KUKA KRL program: EPS_2_251806_MH02A_A_20260212042229.src

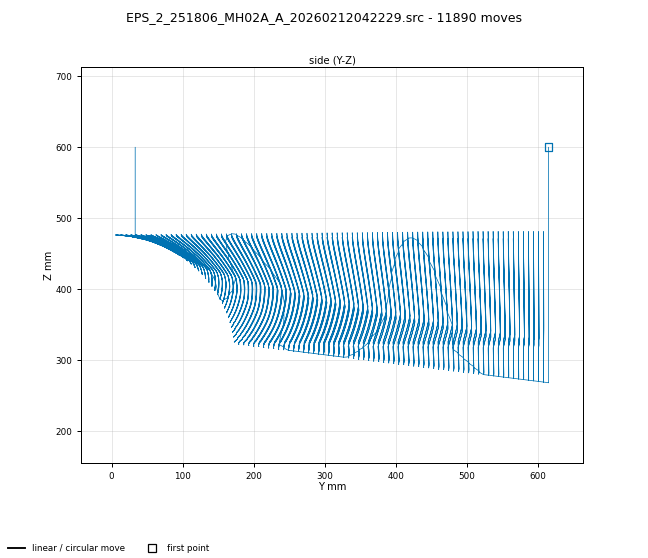
[picture p0: tool path of EPS_2_251806_MH02A_A_20260212042229.src, 11890 of 11892 moves have a stored position in this frame; points joined in program order, loops and branches not executed]
&ACCESS RVP
&REL 4
&COMMENT QRS 19112012
&PARAM EDITMASK = *
DEF PART()
EXT BAS (BAS_COMMAND :IN,REAL :IN )
INT I
BAS (#INITMOV,0 )

;KUKA QRS Post kuka4.cps  Date:22-06-2017 !

File_ID=3010

QRS_PRE_INIT()

;Init var - Until changes are made in qrs_pre_init
Outlet_Square_prg=0
Inlet_1_Square_prg=0
Inlet_2_Square_prg=0
Inlet_3_Square_prg=0
Inlet_4_Square_prg=0
Inlet_5_Square_prg=0

Outlet_1={X 0.000, Y 513.880, Z 332.000, B 0.000, E1 0.000 }
Inlet_1={X 0.000, Y 514.620, Z 322.000, B 0.000, E1 180.000 }
Outlet_1_type=299
Inlet_1_type=299
;QRS#1=Sidecore dimensions
;QRS#2=300-12" PVC SDR 35
;QRS#3=300-12" PVC SDR 35
;QRS#4=
;QRS#5=
;QRS#6=
;QRS#7=
;QRS#8=
;QRS#9=16M PSX
;QRS#10=16M PSX
;QRS#11=
;QRS#12=
;QRS#13=
;QRS#14=
;QRS#15=
;QRS#16=1220x127x762 2,5'
;QRS#17=EPS Height
;QRS#18=481,5
;QRS#19=*
;QRS#20= UPDATED VERSION 22-06-2017
;QRS#21=*
Outlet_Square=0150
Inlet_1_Square=0150
Inlet_2_Square=0
Inlet_3_Square=0
Inlet_4_Square=0
Inlet_5_Square=0
Mill_Square=1
Outlet_Square_Prg=206
Inlet_1_Square_prg=206

QRS_INIT()

$ADVANCE=5

; T1
PTP {E1 173.624,E2 173.624}
PTP {X 0,Y 615.47,A -85,B 0,C 180,E1 173.624,E2 173.624,E3 0,E4 0,E5 0,E6 0}
QRS_SPEED_INIT()
LIN {X 0,Y 615.47,Z 600,A -85,B 0,C 180,E1 173.624,E2 173.624,E3 0,E4 0,E5 0,E6 0} C_VEL
LIN {X 0,Y 615.47,Z 278.503,A -85,B 0,C 180,E1 173.624,E2 173.624} C_VEL
LIN {X 0,Y 615.47,Z 270.325,A -85,B 0,C 180,E1 173.624,E2 173.624} C_VEL
LIN {X 0,Y 615.455,Z 268.325,A -85,B 0,C 180,E1 173.438,E2 173.438} C_VEL
LIN {X 0,Y 615.494,Z 268.326,A -85,B 0,C 180,E1 170.801,E2 170.801} C_VEL
LIN {X 0,Y 615.492,Z 268.318,A -85,B 0,C 180,E1 168.139,E2 168.139} C_VEL
LIN {X 0,Y 615.446,Z 268.325,A -85,B 0,C 180,E1 165.45,E2 165.45} C_VEL
LIN {X 0,Y 615.486,Z 268.318,A -85,B 0,C 180,E1 162.729,E2 162.729} C_VEL
LIN {X 0,Y 615.479,Z 268.326,A -85,B 0,C 180,E1 159.967,E2 159.967} C_VEL
LIN {X 0,Y 615.454,Z 268.324,A -85,B 0,C 180,E1 157.659,E2 157.659} C_VEL
LIN {X 0,Y 615.479,Z 268.319,A -85,B 0,C 180,E1 155.008,E2 155.008} C_VEL
LIN {X 0,Y 615.46,Z 268.325,A -85,B 0,C 180,E1 152.083,E2 152.083} C_VEL
LIN {X 0,Y 615.467,Z 268.322,A -85,B 0,C 180,E1 149.839,E2 149.839} C_VEL
LIN {X 0,Y 615.476,Z 268.322,A -85,B 0,C 180,E1 147.542,E2 147.542} C_VEL
LIN {X 0,Y 615.46,Z 268.325,A -85,B 0,C 180,E1 145.183,E2 145.183} C_VEL
LIN {X 0,Y 615.492,Z 268.316,A -85,B 0,C 180,E1 142.758,E2 142.758} C_VEL
LIN {X 0,Y 615.472,Z 268.324,A -85,B 0,C 180,E1 139.911,E2 139.911} C_VEL
LIN {X 0,Y 615.453,Z 268.325,A -85,B 0,C 180,E1 137.644,E2 137.644} C_VEL
LIN {X 0,Y 615.491,Z 268.315,A -85,B 0,C 180,E1 134.932,E2 134.932} C_VEL
LIN {X 0,Y 615.455,Z 268.324,A -85,B 0,C 180,E1 132.077,E2 132.077} C_VEL
LIN {X 0,Y 615.486,Z 268.547,A -85,B 0,C 180,E1 131.094,E2 131.094} C_VEL
LIN {X 0,Y 615.495,Z 272.375,A -85,B 0,C 180,E1 128.903,E2 128.903} C_VEL
LIN {X 0,Y 615.492,Z 276.811,A -85,B 0,C 180,E1 126.423,E2 126.423} C_VEL
LIN {X 0,Y 615.498,Z 282.132,A -85,B 0,C 180,E1 123.535,E2 123.535} C_VEL
LIN {X 0,Y 615.489,Z 287.143,A -85,B 0,C 180,E1 120.919,E2 120.919} C_VEL
LIN {X 0,Y 615.466,Z 292.012,A -85,B 0,C 180,E1 118.446,E2 118.446} C_VEL
LIN {X 0,Y 615.45,Z 296.042,A -85,B 0,C 180,E1 116.445,E2 116.445} C_VEL
LIN {X 0,Y 615.444,Z 301.065,A -85,B 0,C 180,E1 113.999,E2 113.999} C_VEL
LIN {X 0,Y 615.486,Z 306.417,A -85,B 0,C 180,E1 111.431,E2 111.431} C_VEL
LIN {X 0,Y 615.436,Z 312.479,A -85,B 0,C 180,E1 108.59,E2 108.59} C_VEL
LIN {X 0,Y 615.467,Z 317.53,A -85,B 0,C 180,E1 106.308,E2 106.308} C_VEL
LIN {X 0,Y 615.494,Z 332.686,A -85,B 0,C 180,E1 106.066,E2 106.066} C_VEL
LIN {X 0,Y 615.495,Z 347.732,A -85,B 0,C 180,E1 105.692,E2 105.692} C_VEL
LIN {X 0,Y 615.459,Z 362.612,A -85,B 0,C 180,E1 105.184,E2 105.184} C_VEL
LIN {X 0,Y 615.464,Z 375.186,A -85,B 0,C 180,E1 104.634,E2 104.634} C_VEL
LIN {X 0,Y 615.498,Z 389.266,A -85,B 0,C 180,E1 103.873,E2 103.873} C_VEL
LIN {X 0,Y 615.497,Z 402.017,A -85,B 0,C 180,E1 103.033,E2 103.033} C_VEL
LIN {X 0,Y 615.495,Z 412.714,A -85,B 0,C 180,E1 102.195,E2 102.195} C_VEL
LIN {X 0,Y 615.496,Z 423.542,A -85,B 0,C 180,E1 101.192,E2 101.192} C_VEL
LIN {X 0,Y 615.496,Z 434.059,A -85,B 0,C 180,E1 100.028,E2 100.028} C_VEL
LIN {X 0,Y 615.494,Z 442.802,A -85,B 0,C 180,E1 98.867,E2 98.867} C_VEL
LIN {X 0,Y 615.493,Z 449.121,A -85,B 0,C 180,E1 97.875,E2 97.875} C_VEL
LIN {X 0,Y 615.492,Z 456.054,A -85,B 0,C 180,E1 96.556,E2 96.556} C_VEL
LIN {X 0,Y 615.489,Z 461.499,A -85,B 0,C 180,E1 95.241,E2 95.241} C_VEL
LIN {X 0,Y 615.495,Z 465.62,A -85,B 0,C 180,E1 93.928,E2 93.928} C_VEL
LIN {X 0,Y 615.493,Z 468.526,A -85,B 0,C 180,E1 92.618,E2 92.618} C_VEL
LIN {X 0,Y 615.491,Z 470.276,A -85,B 0,C 180,E1 91.308,E2 91.308} C_VEL
LIN {X 0,Y 615.492,Z 470.885,A -85,B 0,C 180,E1 90,E2 90} C_VEL
LIN {X 0,Y 615.493,Z 470.338,A -85,B 0,C 180,E1 88.691,E2 88.691} C_VEL
LIN {X 0,Y 615.496,Z 468.674,A -85,B 0,C 180,E1 87.382,E2 87.382} C_VEL
LIN {X 0,Y 615.494,Z 465.861,A -85,B 0,C 180,E1 86.071,E2 86.071} C_VEL
LIN {X 0,Y 615.489,Z 461.834,A -85,B 0,C 180,E1 84.759,E2 84.759} C_VEL
LIN {X 0,Y 615.491,Z 456.378,A -85,B 0,C 180,E1 83.42,E2 83.42} C_VEL
LIN {X 0,Y 615.494,Z 449.66,A -85,B 0,C 180,E1 82.124,E2 82.124} C_VEL
LIN {X 0,Y 615.491,Z 441.143,A -85,B 0,C 180,E1 80.801,E2 80.801} C_VEL
LIN {X 0,Y 615.494,Z 432.065,A -85,B 0,C 180,E1 79.639,E2 79.639} C_VEL
LIN {X 0,Y 615.493,Z 422.792,A -85,B 0,C 180,E1 78.64,E2 78.64} C_VEL
LIN {X 0,Y 615.496,Z 410.822,A -85,B 0,C 180,E1 77.554,E2 77.554} C_VEL
LIN {X 0,Y 615.497,Z 398.581,A -85,B 0,C 180,E1 76.631,E2 76.631} C_VEL
LIN {X 0,Y 615.499,Z 385.877,A -85,B 0,C 180,E1 75.834,E2 75.834} C_VEL
LIN {X 0,Y 615.461,Z 371.781,A -85,B 0,C 180,E1 75.112,E2 75.112} C_VEL
LIN {X 0,Y 615.479,Z 357.122,A -85,B 0,C 180,E1 74.519,E2 74.519} C_VEL
LIN {X 0,Y 615.494,Z 342.179,A -85,B 0,C 180,E1 74.063,E2 74.063} C_VEL
LIN {X 0,Y 615.487,Z 326.973,A -85,B 0,C 180,E1 73.738,E2 73.738} C_VEL
LIN {X 0,Y 615.472,Z 317.378,A -85,B 0,C 180,E1 73.591,E2 73.591} C_VEL
LIN {X 0,Y 615.443,Z 312.549,A -85,B 0,C 180,E1 71.353,E2 71.353} C_VEL
LIN {X 0,Y 615.487,Z 306.605,A -85,B 0,C 180,E1 68.568,E2 68.568} C_VEL
LIN {X 0,Y 615.428,Z 300.682,A -85,B 0,C 180,E1 65.726,E2 65.726} C_VEL
LIN {X 0,Y 615.441,Z 296.225,A -85,B 0,C 180,E1 63.554,E2 63.554} C_VEL
LIN {X 0,Y 615.487,Z 290.288,A -85,B 0,C 180,E1 60.594,E2 60.594} C_VEL
LIN {X 0,Y 615.471,Z 285.828,A -85,B 0,C 180,E1 58.314,E2 58.314} C_VEL
LIN {X 0,Y 615.49,Z 281.395,A -85,B 0,C 180,E1 55.979,E2 55.979} C_VEL
LIN {X 0,Y 615.489,Z 276.973,A -85,B 0,C 180,E1 53.576,E2 53.576} C_VEL
LIN {X 0,Y 615.499,Z 272.249,A -85,B 0,C 180,E1 50.937,E2 50.937} C_VEL
LIN {X 0,Y 615.485,Z 268.703,A -85,B 0,C 180,E1 48.906,E2 48.906} C_VEL
LIN {X 0,Y 615.462,Z 268.325,A -85,B 0,C 180,E1 48.525,E2 48.525} C_VEL
LIN {X 0,Y 615.496,Z 268.325,A -85,B 0,C 180,E1 45.852,E2 45.852} C_VEL
LIN {X 0,Y 615.488,Z 268.32,A -85,B 0,C 180,E1 43.048,E2 43.048} C_VEL
LIN {X 0,Y 615.464,Z 268.324,A -85,B 0,C 180,E1 40.087,E2 40.087} C_VEL
LIN {X 0,Y 615.492,Z 268.315,A -85,B 0,C 180,E1 37.242,E2 37.242} C_VEL
LIN {X 0,Y 615.456,Z 268.325,A -85,B 0,C 180,E1 34.697,E2 34.697} C_VEL
LIN {X 0,Y 615.476,Z 268.323,A -85,B 0,C 180,E1 32.33,E2 32.33} C_VEL
LIN {X 0,Y 615.47,Z 268.32,A -85,B 0,C 180,E1 29.793,E2 29.793} C_VEL
LIN {X 0,Y 615.463,Z 268.324,A -85,B 0,C 180,E1 27.042,E2 27.042} C_VEL
LIN {X 0,Y 615.49,Z 268.323,A -85,B 0,C 180,E1 24.272,E2 24.272} C_VEL
LIN {X 0,Y 615.498,Z 268.323,A -85,B 0,C 180,E1 21.432,E2 21.432} C_VEL
LIN {X 0,Y 615.471,Z 268.324,A -85,B 0,C 180,E1 18.602,E2 18.602} C_VEL
LIN {X 0,Y 615.48,Z 268.318,A -85,B 0,C 180,E1 15.905,E2 15.905} C_VEL
LIN {X 0,Y 615.453,Z 268.325,A -85,B 0,C 180,E1 13.202,E2 13.202} C_VEL
LIN {X 0,Y 615.487,Z 268.324,A -85,B 0,C 180,E1 10.527,E2 10.527} C_VEL
LIN {X 0,Y 615.487,Z 268.321,A -85,B 0,C 180,E1 7.876,E2 7.876} C_VEL
LIN {X 0,Y 615.458,Z 268.322,A -85,B 0,C 180,E1 5.242,E2 5.242} C_VEL
LIN {X 0,Y 615.476,Z 268.321,A -85,B 0,C 180,E1 2.618,E2 2.618} C_VEL
LIN {X 0,Y 615.482,Z 268.328,A -85,B 0,C 180,E1 0,E2 0} C_VEL
LIN {X 0,Y 615.47,Z 268.321,A -85,B 0,C 180,E1 -2.618,E2 -2.618} C_VEL
LIN {X 0,Y 615.463,Z 268.322,A -85,B 0,C 180,E1 -5.241,E2 -5.241} C_VEL
LIN {X 0,Y 615.486,Z 268.323,A -85,B 0,C 180,E1 -7.876,E2 -7.876} C_VEL
LIN {X 0,Y 615.483,Z 268.323,A -85,B 0,C 180,E1 -10.527,E2 -10.527} C_VEL
LIN {X 0,Y 615.458,Z 268.323,A -85,B 0,C 180,E1 -13.202,E2 -13.202} C_VEL
LIN {X 0,Y 615.478,Z 268.319,A -85,B 0,C 180,E1 -15.905,E2 -15.905} C_VEL
LIN {X 0,Y 615.478,Z 268.323,A -85,B 0,C 180,E1 -18.646,E2 -18.646} C_VEL
LIN {X 0,Y 615.498,Z 268.325,A -85,B 0,C 180,E1 -21.431,E2 -21.431} C_VEL
LIN {X 0,Y 615.483,Z 268.323,A -85,B 0,C 180,E1 -24.272,E2 -24.272} C_VEL
LIN {X 0,Y 615.466,Z 268.322,A -85,B 0,C 180,E1 -27.042,E2 -27.042} C_VEL
LIN {X 0,Y 615.466,Z 268.321,A -85,B 0,C 180,E1 -29.792,E2 -29.792} C_VEL
LIN {X 0,Y 615.477,Z 268.322,A -85,B 0,C 180,E1 -32.458,E2 -32.458} C_VEL
LIN {X 0,Y 615.459,Z 268.325,A -85,B 0,C 180,E1 -34.817,E2 -34.817} C_VEL
LIN {X 0,Y 615.492,Z 268.316,A -85,B 0,C 180,E1 -37.242,E2 -37.242} C_VEL
LIN {X 0,Y 615.473,Z 268.324,A -85,B 0,C 180,E1 -40.088,E2 -40.088} C_VEL
LIN {X 0,Y 615.452,Z 268.325,A -85,B 0,C 180,E1 -42.356,E2 -42.356} C_VEL
LIN {X 0,Y 615.49,Z 268.315,A -85,B 0,C 180,E1 -45.068,E2 -45.068} C_VEL
LIN {X 0,Y 615.455,Z 268.324,A -85,B 0,C 180,E1 -47.923,E2 -47.923} C_VEL
LIN {X 0,Y 615.48,Z 268.446,A -85,B 0,C 180,E1 -48.81,E2 -48.81} C_VEL
LIN {X 0,Y 615.498,Z 273.148,A -85,B 0,C 180,E1 -51.097,E2 -51.097} C_VEL
LIN {X 0,Y 615.488,Z 278.465,A -85,B 0,C 180,E1 -53.576,E2 -53.576} C_VEL
LIN {X 0,Y 615.494,Z 284.899,A -85,B 0,C 180,E1 -56.465,E2 -56.465} C_VEL
LIN {X 0,Y 615.495,Z 290.877,A -85,B 0,C 180,E1 -59.081,E2 -59.081} C_VEL
LIN {X 0,Y 615.451,Z 296.685,A -85,B 0,C 180,E1 -61.556,E2 -61.556} C_VEL
LIN {X 0,Y 615.438,Z 301.471,A -85,B 0,C 180,E1 -63.554,E2 -63.554} C_VEL
LIN {X 0,Y 615.477,Z 308.525,A -85,B 0,C 180,E1 -66.443,E2 -66.443} C_VEL
LIN {X 0,Y 615.431,Z 315.584,A -85,B 0,C 180,E1 -69.267,E2 -69.267} C_VEL
LIN {X 0,Y 615.494,Z 322.623,A -85,B 0,C 180,E1 -72.043,E2 -72.043} C_VEL
LIN {X 0,Y 615.472,Z 326.699,A -85,B 0,C 180,E1 -73.624,E2 -73.624} C_VEL
LIN {X 0,Y 615.494,Z 344.791,A -85,B 0,C 180,E1 -73.933,E2 -73.933} C_VEL
LIN {X 0,Y 615.495,Z 359.299,A -85,B 0,C 180,E1 -74.307,E2 -74.307} C_VEL
LIN {X 0,Y 615.461,Z 373.789,A -85,B 0,C 180,E1 -74.816,E2 -74.816} C_VEL
LIN {X 0,Y 615.474,Z 387.853,A -85,B 0,C 180,E1 -75.451,E2 -75.451} C_VEL
LIN {X 0,Y 615.496,Z 401.42,A -85,B 0,C 180,E1 -76.21,E2 -76.21} C_VEL
LIN {X 0,Y 615.498,Z 413.79,A -85,B 0,C 180,E1 -77.051,E2 -77.051} C_VEL
LIN {X 0,Y 615.496,Z 425.161,A -85,B 0,C 180,E1 -77.972,E2 -77.972} C_VEL
LIN {X 0,Y 615.498,Z 435.436,A -85,B 0,C 180,E1 -78.957,E2 -78.957} C_VEL
LIN {X 0,Y 615.496,Z 444.421,A -85,B 0,C 180,E1 -79.972,E2 -79.972} C_VEL
LIN {X 0,Y 615.496,Z 453.101,A -85,B 0,C 180,E1 -81.132,E2 -81.132} C_VEL
LIN {X 0,Y 615.494,Z 461.224,A -85,B 0,C 180,E1 -82.454,E2 -82.454} C_VEL
LIN {X 0,Y 615.496,Z 467.729,A -85,B 0,C 180,E1 -83.772,E2 -83.772} C_VEL
LIN {X 0,Y 615.496,Z 472.808,A -85,B 0,C 180,E1 -85.087,E2 -85.087} C_VEL
LIN {X 0,Y 615.495,Z 475.74,A -85,B 0,C 180,E1 -86.071,E2 -86.071} C_VEL
LIN {X 0,Y 615.494,Z 478.6,A -85,B 0,C 180,E1 -87.382,E2 -87.382} C_VEL
LIN {X 0,Y 615.492,Z 480.307,A -85,B 0,C 180,E1 -88.691,E2 -88.691} C_VEL
LIN {X 0,Y 615.491,Z 480.889,A -85,B 0,C 180,E1 -90,E2 -90} C_VEL
LIN {X 0,Y 615.492,Z 480.307,A -85,B 0,C 180,E1 -91.308,E2 -91.308} C_VEL
LIN {X 0,Y 615.494,Z 478.6,A -85,B 0,C 180,E1 -92.618,E2 -92.618} C_VEL
LIN {X 0,Y 615.495,Z 475.741,A -85,B 0,C 180,E1 -93.928,E2 -93.928} C_VEL
LIN {X 0,Y 615.491,Z 471.667,A -85,B 0,C 180,E1 -95.241,E2 -95.241} C_VEL
LIN {X 0,Y 615.49,Z 466.159,A -85,B 0,C 180,E1 -96.58,E2 -96.58} C_VEL
LIN {X 0,Y 615.493,Z 459.395,A -85,B 0,C 180,E1 -97.875,E2 -97.875} C_VEL
LIN {X 0,Y 615.495,Z 450.812,A -85,B 0,C 180,E1 -99.198,E2 -99.198} C_VEL
LIN {X 0,Y 615.494,Z 441.671,A -85,B 0,C 180,E1 -100.36,E2 -100.36} C_VEL
LIN {X 0,Y 615.497,Z 432.358,A -85,B 0,C 180,E1 -101.359,E2 -101.359} C_VEL
LIN {X 0,Y 615.496,Z 421.298,A -85,B 0,C 180,E1 -102.362,E2 -102.362} C_VEL
LIN {X 0,Y 615.498,Z 409.159,A -85,B 0,C 180,E1 -103.285,E2 -103.285} C_VEL
LIN {X 0,Y 615.498,Z 396.407,A -85,B 0,C 180,E1 -104.089,E2 -104.089} C_VEL
LIN {X 0,Y 615.46,Z 382.621,A -85,B 0,C 180,E1 -104.803,E2 -104.803} C_VEL
LIN {X 0,Y 615.474,Z 368.196,A -85,B 0,C 180,E1 -105.395,E2 -105.395} C_VEL
LIN {X 0,Y 615.495,Z 353.267,A -85,B 0,C 180,E1 -105.862,E2 -105.862} C_VEL
LIN {X 0,Y 615.487,Z 338.077,A -85,B 0,C 180,E1 -106.197,E2 -106.197} C_VEL
LIN {X 0,Y 615.472,Z 326.699,A -85,B 0,C 180,E1 -106.376,E2 -106.376} C_VEL
LIN {X 0,Y 615.441,Z 320.876,A -85,B 0,C 180,E1 -108.647,E2 -108.647} C_VEL
LIN {X 0,Y 615.487,Z 313.812,A -85,B 0,C 180,E1 -111.431,E2 -111.431} C_VEL
LIN {X 0,Y 615.426,Z 306.77,A -85,B 0,C 180,E1 -114.274,E2 -114.274} C_VEL
LIN {X 0,Y 615.438,Z 301.472,A -85,B 0,C 180,E1 -116.446,E2 -116.446} C_VEL
LIN {X 0,Y 615.486,Z 294.415,A -85,B 0,C 180,E1 -119.406,E2 -119.406} C_VEL
LIN {X 0,Y 615.467,Z 289.115,A -85,B 0,C 180,E1 -121.686,E2 -121.686} C_VEL
LIN {X 0,Y 615.49,Z 283.803,A -85,B 0,C 180,E1 -124.021,E2 -124.021} C_VEL
LIN {X 0,Y 615.485,Z 278.467,A -85,B 0,C 180,E1 -126.424,E2 -126.424} C_VEL
LIN {X 0,Y 615.496,Z 272.813,A -85,B 0,C 180,E1 -129.063,E2 -129.063} C_VEL
LIN {X 0,Y 615.475,Z 268.324,A -85,B 0,C 180,E1 -131.284,E2 -131.284} C_VEL
LIN {X 0,Y 615.496,Z 268.324,A -85,B 0,C 180,E1 -134.148,E2 -134.148} C_VEL
LIN {X 0,Y 615.488,Z 268.322,A -85,B 0,C 180,E1 -136.951,E2 -136.951} C_VEL
LIN {X 0,Y 615.463,Z 268.321,A -85,B 0,C 180,E1 -139.392,E2 -139.392} C_VEL
LIN {X 0,Y 615.481,Z 268.323,A -85,B 0,C 180,E1 -141.987,E2 -141.987} C_VEL
LIN {X 0,Y 615.459,Z 268.325,A -85,B 0,C 180,E1 -144.382,E2 -144.382} C_VEL
LIN {X 0,Y 615.489,Z 268.318,A -85,B 0,C 180,E1 -146.764,E2 -146.764} C_VEL
LIN {X 0,Y 615.489,Z 268.32,A -85,B 0,C 180,E1 -149.08,E2 -149.08} C_VEL
LIN {X 0,Y 615.447,Z 268.325,A -85,B 0,C 180,E1 -151.554,E2 -151.554} C_VEL
LIN {X 0,Y 615.491,Z 268.317,A -85,B 0,C 180,E1 -154.428,E2 -154.428} C_VEL
LIN {X 0,Y 615.48,Z 268.326,A -85,B 0,C 180,E1 -157.155,E2 -157.155} C_VEL
LIN {X 0,Y 615.446,Z 268.325,A -85,B 0,C 180,E1 -159.45,E2 -159.45} C_VEL
LIN {X 0,Y 615.487,Z 268.318,A -85,B 0,C 180,E1 -162.043,E2 -162.043} C_VEL
LIN {X 0,Y 615.484,Z 268.326,A -85,B 0,C 180,E1 -164.774,E2 -164.774} C_VEL
LIN {X 0,Y 615.469,Z 268.325,A -85,B 0,C 180,E1 -167.47,E2 -167.47} C_VEL
LIN {X 0,Y 615.494,Z 268.314,A -85,B 0,C 180,E1 -170.138,E2 -170.138} C_VEL
LIN {X 0,Y 615.456,Z 268.325,A -85,B 0,C 180,E1 -172.784,E2 -172.784} C_VEL
LIN {X 0,Y 615.495,Z 268.326,A -85,B 0,C 180,E1 -175.416,E2 -175.416} C_VEL
LIN {X 0,Y 615.5,Z 268.315,A -85,B 0,C 180,E1 -178.037,E2 -178.037} C_VEL
LIN {X 0,Y 615.447,Z 268.325,A -85,B 0,C 180,E1 -180.654,E2 -180.654} C_VEL
LIN {X 0,Y 615.487,Z 268.322,A -85,B 0,C 180,E1 -183.273,E2 -183.273} C_VEL
LIN {X 0,Y 615.499,Z 268.319,A -85,B 0,C 180,E1 -185.899,E2 -185.899} C_VEL
LIN {X 0,Y 615.455,Z 268.325,A -85,B 0,C 180,E1 -186.562,E2 -186.562} C_VEL
LIN {X 0,Y 614.784,Z 268.471,A -85,B 0,C 180,E1 -187.108,E2 -187.108} C_VEL
LIN {X 0,Y 611.966,Z 268.881,A -85,B 0,C 180,E1 -187.994,E2 -187.994} C_VEL
LIN {X 0,Y 609.588,Z 269.192,A -85,B 0,C 180,E1 -188.707,E2 -188.707} C_VEL
LIN {X 0,Y 608.556,Z 269.31,A -85,B 0,C 180,E1 -189.257,E2 -189.257} C_VEL
LIN {X 0,Y 608.466,Z 269.318,A -85,B 0,C 180,E1 -189.443,E2 -189.443} C_VEL
LIN {X 0,Y 608.461,Z 269.319,A -85,B 0,C 180,E1 -192,E2 -192} C_VEL
LIN {X 0,Y 608.418,Z 269.321,A -85,B 0,C 180,E1 -194.722,E2 -194.722} C_VEL
LIN {X 0,Y 608.452,Z 269.317,A -85,B 0,C 180,E1 -197.477,E2 -197.477} C_VEL
LIN {X 0,Y 608.44,Z 269.32,A -85,B 0,C 180,E1 -200.275,E2 -200.275} C_VEL
LIN {X 0,Y 608.449,Z 269.318,A -85,B 0,C 180,E1 -202.477,E2 -202.477} C_VEL
LIN {X 0,Y 608.449,Z 269.322,A -85,B 0,C 180,E1 -204.571,E2 -204.571} C_VEL
LIN {X 0,Y 608.467,Z 269.317,A -85,B 0,C 180,E1 -207.207,E2 -207.207} C_VEL
LIN {X 0,Y 608.449,Z 269.317,A -85,B 0,C 180,E1 -209.971,E2 -209.971} C_VEL
LIN {X 0,Y 608.452,Z 269.318,A -85,B 0,C 180,E1 -212.523,E2 -212.523} C_VEL
LIN {X 0,Y 608.425,Z 269.323,A -85,B 0,C 180,E1 -214.904,E2 -214.904} C_VEL
LIN {X 0,Y 608.468,Z 269.316,A -85,B 0,C 180,E1 -217.746,E2 -217.746} C_VEL
LIN {X 0,Y 608.433,Z 269.32,A -85,B 0,C 180,E1 -220.328,E2 -220.328} C_VEL
LIN {X 0,Y 608.452,Z 269.322,A -85,B 0,C 180,E1 -222.96,E2 -222.96} C_VEL
LIN {X 0,Y 608.463,Z 269.32,A -85,B 0,C 180,E1 -225.736,E2 -225.736} C_VEL
LIN {X 0,Y 608.449,Z 269.32,A -85,B 0,C 180,E1 -228.659,E2 -228.659} C_VEL
LIN {X 0,Y 608.48,Z 272.735,A -85,B 0,C 180,E1 -230.702,E2 -230.702} C_VEL
LIN {X 0,Y 608.464,Z 276.956,A -85,B 0,C 180,E1 -233.087,E2 -233.087} C_VEL
LIN {X 0,Y 608.477,Z 281.39,A -85,B 0,C 180,E1 -235.532,E2 -235.532} C_VEL
LIN {X 0,Y 608.438,Z 285.825,A -85,B 0,C 180,E1 -237.905,E2 -237.905} C_VEL
LIN {X 0,Y 608.452,Z 290.297,A -85,B 0,C 180,E1 -240.22,E2 -240.22} C_VEL
LIN {X 0,Y 608.421,Z 296.262,A -85,B 0,C 180,E1 -243.225,E2 -243.225} C_VEL
LIN {X 0,Y 608.388,Z 301.637,A -85,B 0,C 180,E1 -245.867,E2 -245.867} C_VEL
LIN {X 0,Y 608.424,Z 306.7,A -85,B 0,C 180,E1 -248.307,E2 -248.307} C_VEL
LIN {X 0,Y 608.388,Z 313.046,A -85,B 0,C 180,E1 -251.308,E2 -251.308} C_VEL
LIN {X 0,Y 608.394,Z 317.743,A -85,B 0,C 180,E1 -253.495,E2 -253.495} C_VEL
LIN {X 0,Y 608.681,Z 327.53,A -85,B 0,C 180,E1 -253.652,E2 -253.652} C_VEL
LIN {X 0,Y 608.665,Z 342.439,A -85,B 0,C 180,E1 -253.977,E2 -253.977} C_VEL
LIN {X 0,Y 608.611,Z 357.008,A -85,B 0,C 180,E1 -254.427,E2 -254.427} C_VEL
LIN {X 0,Y 608.558,Z 371.685,A -85,B 0,C 180,E1 -255.025,E2 -255.025} C_VEL
LIN {X 0,Y 608.573,Z 385.449,A -85,B 0,C 180,E1 -255.735,E2 -255.735} C_VEL
LIN {X 0,Y 608.547,Z 398.551,A -85,B 0,C 180,E1 -256.561,E2 -256.561} C_VEL
LIN {X 0,Y 608.505,Z 410.846,A -85,B 0,C 180,E1 -257.494,E2 -257.494} C_VEL
LIN {X 0,Y 608.498,Z 422.055,A -85,B 0,C 180,E1 -258.508,E2 -258.508} C_VEL
LIN {X 0,Y 608.477,Z 432.938,A -85,B 0,C 180,E1 -259.687,E2 -259.687} C_VEL
LIN {X 0,Y 608.469,Z 441.987,A -85,B 0,C 180,E1 -260.862,E2 -260.862} C_VEL
LIN {X 0,Y 608.456,Z 449.482,A -85,B 0,C 180,E1 -262.033,E2 -262.033} C_VEL
LIN {X 0,Y 608.445,Z 456.631,A -85,B 0,C 180,E1 -263.397,E2 -263.397} C_VEL
LIN {X 0,Y 608.435,Z 461.995,A -85,B 0,C 180,E1 -264.698,E2 -264.698} C_VEL
LIN {X 0,Y 608.432,Z 466.168,A -85,B 0,C 180,E1 -266.026,E2 -266.026} C_VEL
LIN {X 0,Y 608.421,Z 469.11,A -85,B 0,C 180,E1 -267.352,E2 -267.352} C_VEL
LIN {X 0,Y 608.444,Z 470.881,A -85,B 0,C 180,E1 -268.677,E2 -268.677} C_VEL
LIN {X 0,Y 608.432,Z 471.495,A -85,B 0,C 180,E1 -270,E2 -270} C_VEL
LIN {X 0,Y 608.445,Z 470.944,A -85,B 0,C 180,E1 -271.324,E2 -271.324} C_VEL
LIN {X 0,Y 608.424,Z 469.259,A -85,B 0,C 180,E1 -272.648,E2 -272.648} C_VEL
LIN {X 0,Y 608.431,Z 466.407,A -85,B 0,C 180,E1 -273.974,E2 -273.974} C_VEL
LIN {X 0,Y 608.435,Z 462.328,A -85,B 0,C 180,E1 -275.302,E2 -275.302} C_VEL
LIN {X 0,Y 608.446,Z 456.921,A -85,B 0,C 180,E1 -276.633,E2 -276.633} C_VEL
LIN {X 0,Y 608.457,Z 450.022,A -85,B 0,C 180,E1 -277.967,E2 -277.967} C_VEL
LIN {X 0,Y 608.466,Z 442.59,A -85,B 0,C 180,E1 -279.138,E2 -279.138} C_VEL
LIN {X 0,Y 608.476,Z 433.662,A -85,B 0,C 180,E1 -280.313,E2 -280.313} C_VEL
LIN {X 0,Y 608.495,Z 422.946,A -85,B 0,C 180,E1 -281.492,E2 -281.492} C_VEL
LIN {X 0,Y 608.513,Z 410.905,A -85,B 0,C 180,E1 -282.591,E2 -282.591} C_VEL
LIN {X 0,Y 608.543,Z 398.616,A -85,B 0,C 180,E1 -283.525,E2 -283.525} C_VEL
LIN {X 0,Y 608.588,Z 385.674,A -85,B 0,C 180,E1 -284.342,E2 -284.342} C_VEL
LIN {X 0,Y 608.575,Z 371.769,A -85,B 0,C 180,E1 -285.06,E2 -285.06} C_VEL
LIN {X 0,Y 608.612,Z 357.106,A -85,B 0,C 180,E1 -285.66,E2 -285.66} C_VEL
LIN {X 0,Y 608.662,Z 341.548,A -85,B 0,C 180,E1 -286.138,E2 -286.138} C_VEL
LIN {X 0,Y 608.664,Z 326.29,A -85,B 0,C 180,E1 -286.462,E2 -286.462} C_VEL
LIN {X 0,Y 608.49,Z 318.234,A -85,B 0,C 180,E1 -286.583,E2 -286.583} C_VEL
LIN {X 0,Y 608.405,Z 317.668,A -85,B 0,C 180,E1 -286.63,E2 -286.63} C_VEL
LIN {X 0,Y 608.385,Z 312.855,A -85,B 0,C 180,E1 -288.872,E2 -288.872} C_VEL
LIN {X 0,Y 608.427,Z 306.887,A -85,B 0,C 180,E1 -291.693,E2 -291.693} C_VEL
LIN {X 0,Y 608.387,Z 300.918,A -85,B 0,C 180,E1 -294.574,E2 -294.574} C_VEL
LIN {X 0,Y 608.468,Z 295.574,A -85,B 0,C 180,E1 -297.205,E2 -297.205} C_VEL
LIN {X 0,Y 608.428,Z 290.114,A -85,B 0,C 180,E1 -299.965,E2 -299.965} C_VEL
LIN {X 0,Y 608.464,Z 285.185,A -85,B 0,C 180,E1 -302.522,E2 -302.522} C_VEL
LIN {X 0,Y 608.449,Z 280.08,A -85,B 0,C 180,E1 -305.277,E2 -305.277} C_VEL
LIN {X 0,Y 608.474,Z 275.629,A -85,B 0,C 180,E1 -307.746,E2 -307.746} C_VEL
LIN {X 0,Y 608.482,Z 271.091,A -85,B 0,C 180,E1 -310.332,E2 -310.332} C_VEL
LIN {X 0,Y 608.449,Z 269.366,A -85,B 0,C 180,E1 -311.341,E2 -311.341} C_VEL
LIN {X 0,Y 608.464,Z 269.321,A -85,B 0,C 180,E1 -314.264,E2 -314.264} C_VEL
LIN {X 0,Y 608.451,Z 269.321,A -85,B 0,C 180,E1 -317.04,E2 -317.04} C_VEL
LIN {X 0,Y 608.45,Z 269.317,A -85,B 0,C 180,E1 -319.696,E2 -319.696} C_VEL
LIN {X 0,Y 608.471,Z 269.316,A -85,B 0,C 180,E1 -322.254,E2 -322.254} C_VEL
LIN {X 0,Y 608.43,Z 269.323,A -85,B 0,C 180,E1 -325.096,E2 -325.096} C_VEL
LIN {X 0,Y 608.448,Z 269.318,A -85,B 0,C 180,E1 -327.479,E2 -327.479} C_VEL
LIN {X 0,Y 608.455,Z 269.316,A -85,B 0,C 180,E1 -330.22,E2 -330.22} C_VEL
LIN {X 0,Y 608.467,Z 269.318,A -85,B 0,C 180,E1 -332.794,E2 -332.794} C_VEL
LIN {X 0,Y 608.45,Z 269.321,A -85,B 0,C 180,E1 -335.429,E2 -335.429} C_VEL
LIN {X 0,Y 608.465,Z 269.317,A -85,B 0,C 180,E1 -338.308,E2 -338.308} C_VEL
LIN {X 0,Y 608.46,Z 269.317,A -85,B 0,C 180,E1 -341.285,E2 -341.285} C_VEL
LIN {X 0,Y 608.453,Z 269.317,A -85,B 0,C 180,E1 -343.906,E2 -343.906} C_VEL
LIN {X 0,Y 608.439,Z 269.32,A -85,B 0,C 180,E1 -346.643,E2 -346.643} C_VEL
LIN {X 0,Y 608.463,Z 269.322,A -85,B 0,C 180,E1 -349.35,E2 -349.35} C_VEL
LIN {X 0,Y 608.474,Z 269.316,A -85,B 0,C 180,E1 -352.033,E2 -352.033} C_VEL
LIN {X 0,Y 608.442,Z 269.318,A -85,B 0,C 180,E1 -354.698,E2 -354.698} C_VEL
LIN {X 0,Y 608.468,Z 269.317,A -85,B 0,C 180,E1 -357.352,E2 -357.352} C_VEL
LIN {X 0,Y 608.472,Z 269.32,A -85,B 0,C 180,E1 -360,E2 -360} C_VEL
LIN {X 0,Y 608.463,Z 269.317,A -85,B 0,C 180,E1 -362.648,E2 -362.648} C_VEL
LIN {X 0,Y 608.447,Z 269.318,A -85,B 0,C 180,E1 -365.302,E2 -365.302} C_VEL
LIN {X 0,Y 608.473,Z 269.317,A -85,B 0,C 180,E1 -367.967,E2 -367.967} C_VEL
LIN {X 0,Y 608.463,Z 269.321,A -85,B 0,C 180,E1 -370.65,E2 -370.65} C_VEL
LIN {X 0,Y 608.444,Z 269.319,A -85,B 0,C 180,E1 -373.357,E2 -373.357} C_VEL
LIN {X 0,Y 608.45,Z 269.317,A -85,B 0,C 180,E1 -376.094,E2 -376.094} C_VEL
LIN {X 0,Y 608.45,Z 269.318,A -85,B 0,C 180,E1 -378.87,E2 -378.87} C_VEL
LIN {X 0,Y 608.463,Z 269.319,A -85,B 0,C 180,E1 -381.692,E2 -381.692} C_VEL
LIN {X 0,Y 608.449,Z 269.323,A -85,B 0,C 180,E1 -384.571,E2 -384.571} C_VEL
LIN {X 0,Y 608.468,Z 269.317,A -85,B 0,C 180,E1 -387.207,E2 -387.207} C_VEL
LIN {X 0,Y 608.449,Z 269.317,A -85,B 0,C 180,E1 -389.969,E2 -389.969} C_VEL
LIN {X 0,Y 608.453,Z 269.319,A -85,B 0,C 180,E1 -392.522,E2 -392.522} C_VEL
LIN {X 0,Y 608.424,Z 269.323,A -85,B 0,C 180,E1 -394.903,E2 -394.903} C_VEL
LIN {X 0,Y 608.467,Z 269.316,A -85,B 0,C 180,E1 -397.746,E2 -397.746} C_VEL
LIN {X 0,Y 608.433,Z 269.32,A -85,B 0,C 180,E1 -400.328,E2 -400.328} C_VEL
LIN {X 0,Y 608.452,Z 269.322,A -85,B 0,C 180,E1 -402.96,E2 -402.96} C_VEL
LIN {X 0,Y 608.463,Z 269.32,A -85,B 0,C 180,E1 -405.735,E2 -405.735} C_VEL
LIN {X 0,Y 608.453,Z 269.346,A -85,B 0,C 180,E1 -408.659,E2 -408.659} C_VEL
LIN {X 0,Y 608.481,Z 273.49,A -85,B 0,C 180,E1 -410.701,E2 -410.701} C_VEL
LIN {X 0,Y 608.473,Z 278.521,A -85,B 0,C 180,E1 -413.087,E2 -413.087} C_VEL
LIN {X 0,Y 608.476,Z 283.879,A -85,B 0,C 180,E1 -415.531,E2 -415.531} C_VEL
LIN {X 0,Y 608.451,Z 289.229,A -85,B 0,C 180,E1 -417.905,E2 -417.905} C_VEL
LIN {X 0,Y 608.445,Z 294.547,A -85,B 0,C 180,E1 -420.22,E2 -420.22} C_VEL
LIN {X 0,Y 608.464,Z 300.609,A -85,B 0,C 180,E1 -422.795,E2 -422.795} C_VEL
LIN {X 0,Y 608.386,Z 306.957,A -85,B 0,C 180,E1 -425.426,E2 -425.426} C_VEL
LIN {X 0,Y 608.378,Z 312.275,A -85,B 0,C 180,E1 -427.591,E2 -427.591} C_VEL
LIN {X 0,Y 608.437,Z 319.366,A -85,B 0,C 180,E1 -430.429,E2 -430.429} C_VEL
LIN {X 0,Y 608.422,Z 324.685,A -85,B 0,C 180,E1 -432.523,E2 -432.523} C_VEL
LIN {X 0,Y 608.422,Z 327.035,A -85,B 0,C 180,E1 -433.44,E2 -433.44} C_VEL
LIN {X 0,Y 608.665,Z 334.308,A -85,B 0,C 180,E1 -433.554,E2 -433.554} C_VEL
LIN {X 0,Y 608.66,Z 349.662,A -85,B 0,C 180,E1 -433.862,E2 -433.862} C_VEL
LIN {X 0,Y 608.618,Z 364.497,A -85,B 0,C 180,E1 -434.297,E2 -434.297} C_VEL
LIN {X 0,Y 608.587,Z 378.787,A -85,B 0,C 180,E1 -434.854,E2 -434.854} C_VEL
LIN {X 0,Y 608.568,Z 393.133,A -85,B 0,C 180,E1 -435.564,E2 -435.564} C_VEL
LIN {X 0,Y 608.554,Z 406.664,A -85,B 0,C 180,E1 -436.39,E2 -436.39} C_VEL
LIN {X 0,Y 608.528,Z 419.282,A -85,B 0,C 180,E1 -437.324,E2 -437.324} C_VEL
LIN {X 0,Y 608.498,Z 430.747,A -85,B 0,C 180,E1 -438.339,E2 -438.339} C_VEL
LIN {X 0,Y 608.475,Z 440.387,A -85,B 0,C 180,E1 -439.35,E2 -439.35} C_VEL
LIN {X 0,Y 608.477,Z 449.853,A -85,B 0,C 180,E1 -440.526,E2 -440.526} C_VEL
LIN {X 0,Y 608.456,Z 457.728,A -85,B 0,C 180,E1 -441.698,E2 -441.698} C_VEL
LIN {X 0,Y 608.44,Z 465.087,A -85,B 0,C 180,E1 -443.034,E2 -443.034} C_VEL
LIN {X 0,Y 608.451,Z 470.923,A -85,B 0,C 180,E1 -444.365,E2 -444.365} C_VEL
LIN {X 0,Y 608.427,Z 474.382,A -85,B 0,C 180,E1 -445.362,E2 -445.362} C_VEL
LIN {X 0,Y 608.421,Z 477.885,A -85,B 0,C 180,E1 -446.689,E2 -446.689} C_VEL
LIN {X 0,Y 608.444,Z 480.191,A -85,B 0,C 180,E1 -448.014,E2 -448.014} C_VEL
LIN {X 0,Y 608.434,Z 481.35,A -85,B 0,C 180,E1 -449.338,E2 -449.338} C_VEL
LIN {X 0,Y 608.434,Z 481.351,A -85,B 0,C 180,E1 -450.662,E2 -450.662} C_VEL
LIN {X 0,Y 608.444,Z 480.192,A -85,B 0,C 180,E1 -451.986,E2 -451.986} C_VEL
LIN {X 0,Y 608.421,Z 477.886,A -85,B 0,C 180,E1 -453.311,E2 -453.311} C_VEL
LIN {X 0,Y 608.427,Z 474.384,A -85,B 0,C 180,E1 -454.638,E2 -454.638} C_VEL
LIN {X 0,Y 608.437,Z 469.609,A -85,B 0,C 180,E1 -455.967,E2 -455.967} C_VEL
LIN {X 0,Y 608.456,Z 463.428,A -85,B 0,C 180,E1 -457.299,E2 -457.299} C_VEL
LIN {X 0,Y 608.467,Z 455.656,A -85,B 0,C 180,E1 -458.635,E2 -458.635} C_VEL
LIN {X 0,Y 608.471,Z 447.373,A -85,B 0,C 180,E1 -459.809,E2 -459.809} C_VEL
LIN {X 0,Y 608.492,Z 436.654,A -85,B 0,C 180,E1 -461.063,E2 -461.063} C_VEL
LIN {X 0,Y 608.522,Z 425.279,A -85,B 0,C 180,E1 -462.167,E2 -462.167} C_VEL
LIN {X 0,Y 608.547,Z 413.86,A -85,B 0,C 180,E1 -463.099,E2 -463.099} C_VEL
LIN {X 0,Y 608.561,Z 401.455,A -85,B 0,C 180,E1 -463.95,E2 -463.95} C_VEL
LIN {X 0,Y 608.575,Z 387.869,A -85,B 0,C 180,E1 -464.718,E2 -464.718} C_VEL
LIN {X 0,Y 608.593,Z 373.804,A -85,B 0,C 180,E1 -465.359,E2 -465.359} C_VEL
LIN {X 0,Y 608.643,Z 359.318,A -85,B 0,C 180,E1 -465.873,E2 -465.873} C_VEL
LIN {X 0,Y 608.682,Z 344.1,A -85,B 0,C 180,E1 -466.268,E2 -466.268} C_VEL
LIN {X 0,Y 608.514,Z 327.673,A -85,B 0,C 180,E1 -466.544,E2 -466.544} C_VEL
LIN {X 0,Y 608.403,Z 327.025,A -85,B 0,C 180,E1 -466.564,E2 -466.564} C_VEL
LIN {X 0,Y 608.41,Z 321.14,A -85,B 0,C 180,E1 -468.87,E2 -468.87} C_VEL
LIN {X 0,Y 608.426,Z 314.049,A -85,B 0,C 180,E1 -471.692,E2 -471.692} C_VEL
LIN {X 0,Y 608.41,Z 308.017,A -85,B 0,C 180,E1 -474.138,E2 -474.138} C_VEL
LIN {X 0,Y 608.42,Z 301.64,A -85,B 0,C 180,E1 -476.775,E2 -476.775} C_VEL
LIN {X 0,Y 608.431,Z 296.321,A -85,B 0,C 180,E1 -479.021,E2 -479.021} C_VEL
LIN {X 0,Y 608.474,Z 291.003,A -85,B 0,C 180,E1 -481.315,E2 -481.315} C_VEL
LIN {X 0,Y 608.479,Z 285.514,A -85,B 0,C 180,E1 -483.736,E2 -483.736} C_VEL
LIN {X 0,Y 608.476,Z 280.304,A -85,B 0,C 180,E1 -486.089,E2 -486.089} C_VEL
LIN {X 0,Y 608.475,Z 274.971,A -85,B 0,C 180,E1 -488.587,E2 -488.587} C_VEL
LIN {X 0,Y 608.507,Z 269.68,A -85,B 0,C 180,E1 -491.171,E2 -491.171} C_VEL
LIN {X 0,Y 608.455,Z 269.319,A -85,B 0,C 180,E1 -491.476,E2 -491.476} C_VEL
LIN {X 0,Y 608.464,Z 269.32,A -85,B 0,C 180,E1 -494.265,E2 -494.265} C_VEL
LIN {X 0,Y 608.45,Z 269.322,A -85,B 0,C 180,E1 -497.04,E2 -497.04} C_VEL
LIN {X 0,Y 608.445,Z 269.318,A -85,B 0,C 180,E1 -499.696,E2 -499.696} C_VEL
LIN {X 0,Y 608.467,Z 269.316,A -85,B 0,C 180,E1 -502.254,E2 -502.254} C_VEL
LIN {X 0,Y 608.425,Z 269.323,A -85,B 0,C 180,E1 -505.096,E2 -505.096} C_VEL
LIN {X 0,Y 608.452,Z 269.319,A -85,B 0,C 180,E1 -507.477,E2 -507.477} C_VEL
LIN {X 0,Y 608.452,Z 269.317,A -85,B 0,C 180,E1 -510.22,E2 -510.22} C_VEL
LIN {X 0,Y 608.467,Z 269.317,A -85,B 0,C 180,E1 -512.793,E2 -512.793} C_VEL
LIN {X 0,Y 608.449,Z 269.323,A -85,B 0,C 180,E1 -515.429,E2 -515.429} C_VEL
LIN {X 0,Y 608.463,Z 269.318,A -85,B 0,C 180,E1 -518.308,E2 -518.308} C_VEL
LIN {X 0,Y 608.462,Z 269.318,A -85,B 0,C 180,E1 -521.283,E2 -521.283} C_VEL
LIN {X 0,Y 608.45,Z 269.317,A -85,B 0,C 180,E1 -523.906,E2 -523.906} C_VEL
LIN {X 0,Y 608.442,Z 269.319,A -85,B 0,C 180,E1 -526.643,E2 -526.643} C_VEL
LIN {X 0,Y 608.463,Z 269.321,A -85,B 0,C 180,E1 -529.35,E2 -529.35} C_VEL
LIN {X 0,Y 608.473,Z 269.316,A -85,B 0,C 180,E1 -532.033,E2 -532.033} C_VEL
LIN {X 0,Y 608.445,Z 269.318,A -85,B 0,C 180,E1 -534.698,E2 -534.698} C_VEL
LIN {X 0,Y 608.465,Z 269.317,A -85,B 0,C 180,E1 -537.352,E2 -537.352} C_VEL
LIN {X 0,Y 608.469,Z 269.321,A -85,B 0,C 180,E1 -540,E2 -540} C_VEL
LIN {X 0,Y 608.465,Z 269.317,A -85,B 0,C 180,E1 -542.648,E2 -542.648} C_VEL
LIN {X 0,Y 608.444,Z 269.318,A -85,B 0,C 180,E1 -545.302,E2 -545.302} C_VEL
LIN {X 0,Y 608.473,Z 269.316,A -85,B 0,C 180,E1 -547.967,E2 -547.967} C_VEL
LIN {X 0,Y 608.466,Z 269.318,A -85,B 0,C 180,E1 -549.443,E2 -549.443} C_VEL
LIN {X 0,Y 607.785,Z 269.4,A -85,B 0,C 180,E1 -549.995,E2 -549.995} C_VEL
LIN {X 0,Y 604.932,Z 269.759,A -85,B 0,C 180,E1 -550.892,E2 -550.892} C_VEL
LIN {X 0,Y 602.526,Z 270.061,A -85,B 0,C 180,E1 -551.613,E2 -551.613} C_VEL
LIN {X 0,Y 601.488,Z 270.19,A -85,B 0,C 180,E1 -552.17,E2 -552.17} C_VEL
LIN {X 0,Y 601.4,Z 270.198,A -85,B 0,C 180,E1 -552.358,E2 -552.358} C_VEL
LIN {X 0,Y 601.391,Z 270.198,A -85,B 0,C 180,E1 -554.898,E2 -554.898} C_VEL
LIN {X 0,Y 601.427,Z 270.196,A -85,B 0,C 180,E1 -556.986,E2 -556.986} C_VEL
LIN {X 0,Y 601.394,Z 270.201,A -85,B 0,C 180,E1 -559.81,E2 -559.81} C_VEL
LIN {X 0,Y 601.404,Z 270.198,A -85,B 0,C 180,E1 -562.683,E2 -562.683} C_VEL
LIN {X 0,Y 601.4,Z 270.197,A -85,B 0,C 180,E1 -564.879,E2 -564.879} C_VEL
LIN {X 0,Y 601.403,Z 270.199,A -85,B 0,C 180,E1 -567.362,E2 -567.362} C_VEL
LIN {X 0,Y 601.419,Z 270.194,A -85,B 0,C 180,E1 -570.165,E2 -570.165} C_VEL
LIN {X 0,Y 601.415,Z 270.194,A -85,B 0,C 180,E1 -572.716,E2 -572.716} C_VEL
LIN {X 0,Y 601.374,Z 270.204,A -85,B 0,C 180,E1 -575.111,E2 -575.111} C_VEL
LIN {X 0,Y 601.432,Z 270.191,A -85,B 0,C 180,E1 -577.419,E2 -577.419} C_VEL
LIN {X 0,Y 601.408,Z 270.198,A -85,B 0,C 180,E1 -579.995,E2 -579.995} C_VEL
LIN {X 0,Y 601.401,Z 270.199,A -85,B 0,C 180,E1 -582.671,E2 -582.671} C_VEL
LIN {X 0,Y 601.421,Z 270.194,A -85,B 0,C 180,E1 -585.483,E2 -585.483} C_VEL
LIN {X 0,Y 601.41,Z 270.195,A -85,B 0,C 180,E1 -588.409,E2 -588.409} C_VEL
LIN {X 0,Y 601.432,Z 271.504,A -85,B 0,C 180,E1 -589.425,E2 -589.425} C_VEL
LIN {X 0,Y 601.432,Z 275.486,A -85,B 0,C 180,E1 -591.734,E2 -591.734} C_VEL
LIN {X 0,Y 601.41,Z 279.947,A -85,B 0,C 180,E1 -594.248,E2 -594.248} C_VEL
LIN {X 0,Y 601.414,Z 284.37,A -85,B 0,C 180,E1 -596.687,E2 -596.687} C_VEL
LIN {X 0,Y 601.367,Z 288.808,A -85,B 0,C 180,E1 -599.056,E2 -599.056} C_VEL
LIN {X 0,Y 601.398,Z 293.281,A -85,B 0,C 180,E1 -601.372,E2 -601.372} C_VEL
LIN {X 0,Y 601.37,Z 298.766,A -85,B 0,C 180,E1 -604.142,E2 -604.142} C_VEL
LIN {X 0,Y 601.343,Z 303.718,A -85,B 0,C 180,E1 -606.587,E2 -606.587} C_VEL
LIN {X 0,Y 601.3,Z 309.683,A -85,B 0,C 180,E1 -609.474,E2 -609.474} C_VEL
LIN {X 0,Y 601.349,Z 315.648,A -85,B 0,C 180,E1 -612.311,E2 -612.311} C_VEL
LIN {X 0,Y 601.315,Z 317.75,A -85,B 0,C 180,E1 -613.297,E2 -613.297} C_VEL
LIN {X 0,Y 601.86,Z 321.471,A -85,B 0,C 180,E1 -613.366,E2 -613.366} C_VEL
LIN {X 0,Y 601.855,Z 337.349,A -85,B 0,C 180,E1 -613.665,E2 -613.665} C_VEL
LIN {X 0,Y 601.763,Z 353.177,A -85,B 0,C 180,E1 -614.114,E2 -614.114} C_VEL
LIN {X 0,Y 601.694,Z 367.779,A -85,B 0,C 180,E1 -614.677,E2 -614.677} C_VEL
LIN {X 0,Y 601.639,Z 381.861,A -85,B 0,C 180,E1 -615.368,E2 -615.368} C_VEL
LIN {X 0,Y 601.621,Z 395.775,A -85,B 0,C 180,E1 -616.215,E2 -616.215} C_VEL
LIN {X 0,Y 601.531,Z 408.735,A -85,B 0,C 180,E1 -617.175,E2 -617.175} C_VEL
LIN {X 0,Y 601.489,Z 420.285,A -85,B 0,C 180,E1 -618.202,E2 -618.202} C_VEL
LIN {X 0,Y 601.43,Z 429.999,A -85,B 0,C 180,E1 -619.225,E2 -619.225} C_VEL
LIN {X 0,Y 601.428,Z 439.529,A -85,B 0,C 180,E1 -620.415,E2 -620.415} C_VEL
LIN {X 0,Y 601.377,Z 447.463,A -85,B 0,C 180,E1 -621.601,E2 -621.601} C_VEL
LIN {X 0,Y 601.368,Z 454.874,A -85,B 0,C 180,E1 -622.952,E2 -622.952} C_VEL
LIN {X 0,Y 601.373,Z 460.76,A -85,B 0,C 180,E1 -624.299,E2 -624.299} C_VEL
LIN {X 0,Y 601.327,Z 464.242,A -85,B 0,C 180,E1 -625.308,E2 -625.308} C_VEL
LIN {X 0,Y 601.336,Z 467.79,A -85,B 0,C 180,E1 -626.65,E2 -626.65} C_VEL
LIN {X 0,Y 601.343,Z 470.14,A -85,B 0,C 180,E1 -627.991,E2 -627.991} C_VEL
LIN {X 0,Y 601.334,Z 471.337,A -85,B 0,C 180,E1 -629.331,E2 -629.331} C_VEL
LIN {X 0,Y 601.335,Z 471.361,A -85,B 0,C 180,E1 -630.67,E2 -630.67} C_VEL
LIN {X 0,Y 601.343,Z 470.244,A -85,B 0,C 180,E1 -632.01,E2 -632.01} C_VEL
LIN {X 0,Y 601.339,Z 467.982,A -85,B 0,C 180,E1 -633.35,E2 -633.35} C_VEL
LIN {X 0,Y 601.328,Z 464.524,A -85,B 0,C 180,E1 -634.693,E2 -634.693} C_VEL
LIN {X 0,Y 601.358,Z 459.797,A -85,B 0,C 180,E1 -636.038,E2 -636.038} C_VEL
LIN {X 0,Y 601.366,Z 453.666,A -85,B 0,C 180,E1 -637.386,E2 -637.386} C_VEL
LIN {X 0,Y 601.389,Z 445.95,A -85,B 0,C 180,E1 -638.738,E2 -638.738} C_VEL
LIN {X 0,Y 601.428,Z 437.706,A -85,B 0,C 180,E1 -639.925,E2 -639.925} C_VEL
LIN {X 0,Y 601.443,Z 427.365,A -85,B 0,C 180,E1 -641.164,E2 -641.164} C_VEL
LIN {X 0,Y 601.501,Z 415.784,A -85,B 0,C 180,E1 -642.312,E2 -642.312} C_VEL
LIN {X 0,Y 601.557,Z 404.462,A -85,B 0,C 180,E1 -643.255,E2 -643.255} C_VEL
LIN {X 0,Y 601.624,Z 391.312,A -85,B 0,C 180,E1 -644.168,E2 -644.168} C_VEL
LIN {X 0,Y 601.665,Z 378.758,A -85,B 0,C 180,E1 -644.891,E2 -644.891} C_VEL
LIN {X 0,Y 601.708,Z 364.879,A -85,B 0,C 180,E1 -645.54,E2 -645.54} C_VEL
LIN {X 0,Y 601.802,Z 350.659,A -85,B 0,C 180,E1 -646.059,E2 -646.059} C_VEL
LIN {X 0,Y 601.862,Z 335.414,A -85,B 0,C 180,E1 -646.471,E2 -646.471} C_VEL
LIN {X 0,Y 601.817,Z 320.077,A -85,B 0,C 180,E1 -646.745,E2 -646.745} C_VEL
LIN {X 0,Y 601.317,Z 317.718,A -85,B 0,C 180,E1 -646.807,E2 -646.807} C_VEL
LIN {X 0,Y 601.303,Z 312.854,A -85,B 0,C 180,E1 -649.103,E2 -649.103} C_VEL
LIN {X 0,Y 601.32,Z 306.886,A -85,B 0,C 180,E1 -651.963,E2 -651.963} C_VEL
LIN {X 0,Y 601.322,Z 302.161,A -85,B 0,C 180,E1 -654.268,E2 -654.268} C_VEL
LIN {X 0,Y 601.403,Z 296.44,A -85,B 0,C 180,E1 -657.113,E2 -657.113} C_VEL
LIN {X 0,Y 601.375,Z 291.963,A -85,B 0,C 180,E1 -659.395,E2 -659.395} C_VEL
LIN {X 0,Y 601.433,Z 286.026,A -85,B 0,C 180,E1 -662.515,E2 -662.515} C_VEL
LIN {X 0,Y 601.416,Z 281.258,A -85,B 0,C 180,E1 -665.114,E2 -665.114} C_VEL
LIN {X 0,Y 601.438,Z 277.132,A -85,B 0,C 180,E1 -667.418,E2 -667.418} C_VEL
LIN {X 0,Y 601.422,Z 272.646,A -85,B 0,C 180,E1 -669.994,E2 -669.994} C_VEL
LIN {X 0,Y 601.41,Z 270.197,A -85,B 0,C 180,E1 -671.591,E2 -671.591} C_VEL
LIN {X 0,Y 601.423,Z 270.195,A -85,B 0,C 180,E1 -674.535,E2 -674.535} C_VEL
LIN {X 0,Y 601.401,Z 270.199,A -85,B 0,C 180,E1 -677.41,E2 -677.41} C_VEL
LIN {X 0,Y 601.443,Z 270.194,A -85,B 0,C 180,E1 -680.463,E2 -680.463} C_VEL
LIN {X 0,Y 601.403,Z 270.201,A -85,B 0,C 180,E1 -683.417,E2 -683.417} C_VEL
LIN {X 0,Y 601.425,Z 270.194,A -85,B 0,C 180,E1 -686.064,E2 -686.064} C_VEL
LIN {X 0,Y 601.427,Z 270.193,A -85,B 0,C 180,E1 -689.058,E2 -689.058} C_VEL
LIN {X 0,Y 601.409,Z 270.196,A -85,B 0,C 180,E1 -691.372,E2 -691.372} C_VEL
LIN {X 0,Y 601.411,Z 270.199,A -85,B 0,C 180,E1 -694.132,E2 -694.132} C_VEL
LIN {X 0,Y 601.419,Z 270.194,A -85,B 0,C 180,E1 -696.59,E2 -696.59} C_VEL
LIN {X 0,Y 601.404,Z 270.195,A -85,B 0,C 180,E1 -699.477,E2 -699.477} C_VEL
LIN {X 0,Y 601.396,Z 270.196,A -85,B 0,C 180,E1 -702.312,E2 -702.312} C_VEL
LIN {X 0,Y 601.413,Z 270.196,A -85,B 0,C 180,E1 -704.409,E2 -704.409} C_VEL
LIN {X 0,Y 601.396,Z 270.196,A -85,B 0,C 180,E1 -707.171,E2 -707.171} C_VEL
LIN {X 0,Y 601.438,Z 270.191,A -85,B 0,C 180,E1 -709.905,E2 -709.905} C_VEL
LIN {X 0,Y 601.399,Z 270.199,A -85,B 0,C 180,E1 -712.614,E2 -712.614} C_VEL
LIN {X 0,Y 601.425,Z 270.196,A -85,B 0,C 180,E1 -715.308,E2 -715.308} C_VEL
LIN {X 0,Y 601.436,Z 270.191,A -85,B 0,C 180,E1 -717.991,E2 -717.991} C_VEL
LIN {X 0,Y 601.42,Z 270.193,A -85,B 0,C 180,E1 -720.669,E2 -720.669} C_VEL
LIN {X 0,Y 601.434,Z 270.194,A -85,B 0,C 180,E1 -723.349,E2 -723.349} C_VEL
LIN {X 0,Y 601.435,Z 270.196,A -85,B 0,C 180,E1 -726.037,E2 -726.037} C_VEL
LIN {X 0,Y 601.399,Z 270.196,A -85,B 0,C 180,E1 -728.738,E2 -728.738} C_VEL
LIN {X 0,Y 601.431,Z 270.191,A -85,B 0,C 180,E1 -731.458,E2 -731.458} C_VEL
LIN {X 0,Y 601.408,Z 270.196,A -85,B 0,C 180,E1 -734.206,E2 -734.206} C_VEL
LIN {X 0,Y 601.428,Z 270.196,A -85,B 0,C 180,E1 -736.986,E2 -736.986} C_VEL
LIN {X 0,Y 601.396,Z 270.201,A -85,B 0,C 180,E1 -739.81,E2 -739.81} C_VEL
LIN {X 0,Y 601.403,Z 270.197,A -85,B 0,C 180,E1 -742.683,E2 -742.683} C_VEL
LIN {X 0,Y 601.4,Z 270.197,A -85,B 0,C 180,E1 -744.879,E2 -744.879} C_VEL
LIN {X 0,Y 601.404,Z 270.198,A -85,B 0,C 180,E1 -747.361,E2 -747.361} C_VEL
LIN {X 0,Y 601.402,Z 270.196,A -85,B 0,C 180,E1 -750.165,E2 -750.165} C_VEL
LIN {X 0,Y 601.417,Z 270.194,A -85,B 0,C 180,E1 -752.716,E2 -752.716} C_VEL
LIN {X 0,Y 601.374,Z 270.204,A -85,B 0,C 180,E1 -755.11,E2 -755.11} C_VEL
LIN {X 0,Y 601.434,Z 270.191,A -85,B 0,C 180,E1 -757.419,E2 -757.419} C_VEL
LIN {X 0,Y 601.41,Z 270.198,A -85,B 0,C 180,E1 -759.995,E2 -759.995} C_VEL
LIN {X 0,Y 601.402,Z 270.199,A -85,B 0,C 180,E1 -762.671,E2 -762.671} C_VEL
LIN {X 0,Y 601.424,Z 270.194,A -85,B 0,C 180,E1 -765.482,E2 -765.482} C_VEL
LIN {X 0,Y 601.436,Z 270.237,A -85,B 0,C 180,E1 -768.527,E2 -768.527} C_VEL
LIN {X 0,Y 601.473,Z 274.964,A -85,B 0,C 180,E1 -770.879,E2 -770.879} C_VEL
LIN {X 0,Y 601.447,Z 280.945,A -85,B 0,C 180,E1 -773.733,E2 -773.733} C_VEL
LIN {X 0,Y 601.437,Z 286.036,A -85,B 0,C 180,E1 -776.064,E2 -776.064} C_VEL
LIN {X 0,Y 601.439,Z 291.601,A -85,B 0,C 180,E1 -778.542,E2 -778.542} C_VEL
LIN {X 0,Y 601.41,Z 298.093,A -85,B 0,C 180,E1 -781.372,E2 -781.372} C_VEL
LIN {X 0,Y 601.367,Z 304.616,A -85,B 0,C 180,E1 -784.142,E2 -784.142} C_VEL
LIN {X 0,Y 601.36,Z 310.502,A -85,B 0,C 180,E1 -786.587,E2 -786.587} C_VEL
LIN {X 0,Y 601.32,Z 317.594,A -85,B 0,C 180,E1 -789.474,E2 -789.474} C_VEL
LIN {X 0,Y 601.346,Z 322.912,A -85,B 0,C 180,E1 -791.606,E2 -791.606} C_VEL
LIN {X 0,Y 601.336,Z 327.027,A -85,B 0,C 180,E1 -793.236,E2 -793.236} C_VEL
LIN {X 0,Y 601.89,Z 331.195,A -85,B 0,C 180,E1 -793.318,E2 -793.318} C_VEL
LIN {X 0,Y 601.846,Z 345.765,A -85,B 0,C 180,E1 -793.582,E2 -793.582} C_VEL
LIN {X 0,Y 601.793,Z 360.615,A -85,B 0,C 180,E1 -793.984,E2 -793.984} C_VEL
LIN {X 0,Y 601.72,Z 374.842,A -85,B 0,C 180,E1 -794.504,E2 -794.504} C_VEL
LIN {X 0,Y 601.676,Z 389.527,A -85,B 0,C 180,E1 -795.196,E2 -795.196} C_VEL
LIN {X 0,Y 601.606,Z 403.076,A -85,B 0,C 180,E1 -795.988,E2 -795.988} C_VEL
LIN {X 0,Y 601.539,Z 416.101,A -85,B 0,C 180,E1 -796.917,E2 -796.917} C_VEL
LIN {X 0,Y 601.514,Z 427.191,A -85,B 0,C 180,E1 -797.859,E2 -797.859} C_VEL
LIN {X 0,Y 601.437,Z 438.274,A -85,B 0,C 180,E1 -798.982,E2 -798.982} C_VEL
LIN {X 0,Y 601.427,Z 447.369,A -85,B 0,C 180,E1 -800.075,E2 -800.075} C_VEL
LIN {X 0,Y 601.388,Z 455.653,A -85,B 0,C 180,E1 -801.262,E2 -801.262} C_VEL
LIN {X 0,Y 601.365,Z 463.425,A -85,B 0,C 180,E1 -802.614,E2 -802.614} C_VEL
LIN {X 0,Y 601.357,Z 469.607,A -85,B 0,C 180,E1 -803.962,E2 -803.962} C_VEL
LIN {X 0,Y 601.33,Z 474.383,A -85,B 0,C 180,E1 -805.307,E2 -805.307} C_VEL
LIN {X 0,Y 601.337,Z 477.886,A -85,B 0,C 180,E1 -806.65,E2 -806.65} C_VEL
LIN {X 0,Y 601.343,Z 480.192,A -85,B 0,C 180,E1 -807.99,E2 -807.99} C_VEL
LIN {X 0,Y 601.335,Z 481.35,A -85,B 0,C 180,E1 -809.33,E2 -809.33} C_VEL
LIN {X 0,Y 601.335,Z 481.35,A -85,B 0,C 180,E1 -810.669,E2 -810.669} C_VEL
LIN {X 0,Y 601.343,Z 480.192,A -85,B 0,C 180,E1 -812.009,E2 -812.009} C_VEL
LIN {X 0,Y 601.337,Z 477.886,A -85,B 0,C 180,E1 -813.35,E2 -813.35} C_VEL
LIN {X 0,Y 601.33,Z 474.384,A -85,B 0,C 180,E1 -814.692,E2 -814.692} C_VEL
LIN {X 0,Y 601.357,Z 469.609,A -85,B 0,C 180,E1 -816.037,E2 -816.037} C_VEL
LIN {X 0,Y 601.365,Z 463.427,A -85,B 0,C 180,E1 -817.386,E2 -817.386} C_VEL
LIN {X 0,Y 601.388,Z 455.656,A -85,B 0,C 180,E1 -818.738,E2 -818.738} C_VEL
LIN {X 0,Y 601.427,Z 447.373,A -85,B 0,C 180,E1 -819.925,E2 -819.925} C_VEL
LIN {X 0,Y 601.46,Z 436.935,A -85,B 0,C 180,E1 -821.164,E2 -821.164} C_VEL
LIN {X 0,Y 601.513,Z 427.197,A -85,B 0,C 180,E1 -822.14,E2 -822.14} C_VEL
LIN {X 0,Y 601.57,Z 415.022,A -85,B 0,C 180,E1 -823.168,E2 -823.168} C_VEL
LIN {X 0,Y 601.605,Z 403.085,A -85,B 0,C 180,E1 -824.011,E2 -824.011} C_VEL
LIN {X 0,Y 601.675,Z 389.536,A -85,B 0,C 180,E1 -824.804,E2 -824.804} C_VEL
LIN {X 0,Y 601.719,Z 374.854,A -85,B 0,C 180,E1 -825.496,E2 -825.496} C_VEL
LIN {X 0,Y 601.804,Z 360.633,A -85,B 0,C 180,E1 -826.015,E2 -826.015} C_VEL
LIN {X 0,Y 601.857,Z 345.781,A -85,B 0,C 180,E1 -826.418,E2 -826.418} C_VEL
LIN {X 0,Y 601.869,Z 331.042,A -85,B 0,C 180,E1 -826.685,E2 -826.685} C_VEL
LIN {X 0,Y 601.328,Z 327.028,A -85,B 0,C 180,E1 -826.764,E2 -826.764} C_VEL
LIN {X 0,Y 601.357,Z 321.14,A -85,B 0,C 180,E1 -829.1,E2 -829.1} C_VEL
LIN {X 0,Y 601.329,Z 314.049,A -85,B 0,C 180,E1 -831.962,E2 -831.962} C_VEL
LIN {X 0,Y 601.342,Z 308.422,A -85,B 0,C 180,E1 -834.273,E2 -834.273} C_VEL
LIN {X 0,Y 601.361,Z 303.413,A -85,B 0,C 180,E1 -836.365,E2 -836.365} C_VEL
LIN {X 0,Y 601.413,Z 297.728,A -85,B 0,C 180,E1 -838.785,E2 -838.785} C_VEL
LIN {X 0,Y 601.407,Z 290.997,A -85,B 0,C 180,E1 -841.726,E2 -841.726} C_VEL
LIN {X 0,Y 601.433,Z 285.636,A -85,B 0,C 180,E1 -844.117,E2 -844.117} C_VEL
LIN {X 0,Y 601.445,Z 280.278,A -85,B 0,C 180,E1 -846.579,E2 -846.579} C_VEL
LIN {X 0,Y 601.472,Z 274.965,A -85,B 0,C 180,E1 -849.121,E2 -849.121} C_VEL
LIN {X 0,Y 601.426,Z 270.196,A -85,B 0,C 180,E1 -851.504,E2 -851.504} C_VEL
LIN {X 0,Y 601.444,Z 270.191,A -85,B 0,C 180,E1 -853.584,E2 -853.584} C_VEL
LIN {X 0,Y 601.422,Z 270.193,A -85,B 0,C 180,E1 -856.427,E2 -856.427} C_VEL
LIN {X 0,Y 601.404,Z 270.195,A -85,B 0,C 180,E1 -859.427,E2 -859.427} C_VEL
LIN {X 0,Y 601.42,Z 270.199,A -85,B 0,C 180,E1 -861.732,E2 -861.732} C_VEL
LIN {X 0,Y 601.369,Z 270.2,A -85,B 0,C 180,E1 -864.244,E2 -864.244} C_VEL
LIN {X 0,Y 601.423,Z 270.195,A -85,B 0,C 180,E1 -866.686,E2 -866.686} C_VEL
LIN {X 0,Y 601.425,Z 270.195,A -85,B 0,C 180,E1 -869.058,E2 -869.058} C_VEL
LIN {X 0,Y 601.405,Z 270.196,A -85,B 0,C 180,E1 -871.372,E2 -871.372} C_VEL
LIN {X 0,Y 601.389,Z 270.199,A -85,B 0,C 180,E1 -873.636,E2 -873.636} C_VEL
LIN {X 0,Y 601.416,Z 270.194,A -85,B 0,C 180,E1 -876.59,E2 -876.59} C_VEL
LIN {X 0,Y 601.402,Z 270.195,A -85,B 0,C 180,E1 -879.477,E2 -879.477} C_VEL
LIN {X 0,Y 601.396,Z 270.196,A -85,B 0,C 180,E1 -882.312,E2 -882.312} C_VEL
LIN {X 0,Y 601.409,Z 270.197,A -85,B 0,C 180,E1 -884.409,E2 -884.409} C_VEL
LIN {X 0,Y 601.401,Z 270.196,A -85,B 0,C 180,E1 -887.171,E2 -887.171} C_VEL
LIN {X 0,Y 601.437,Z 270.191,A -85,B 0,C 180,E1 -889.905,E2 -889.905} C_VEL
LIN {X 0,Y 601.395,Z 270.199,A -85,B 0,C 180,E1 -892.614,E2 -892.614} C_VEL
LIN {X 0,Y 601.426,Z 270.197,A -85,B 0,C 180,E1 -895.308,E2 -895.308} C_VEL
LIN {X 0,Y 601.436,Z 270.192,A -85,B 0,C 180,E1 -897.991,E2 -897.991} C_VEL
LIN {X 0,Y 601.418,Z 270.193,A -85,B 0,C 180,E1 -900.67,E2 -900.67} C_VEL
LIN {X 0,Y 601.431,Z 270.194,A -85,B 0,C 180,E1 -903.35,E2 -903.35} C_VEL
LIN {X 0,Y 601.434,Z 270.196,A -85,B 0,C 180,E1 -906.037,E2 -906.037} C_VEL
LIN {X 0,Y 601.4,Z 270.196,A -85,B 0,C 180,E1 -908.738,E2 -908.738} C_VEL
LIN {X 0,Y 601.428,Z 270.192,A -85,B 0,C 180,E1 -911.458,E2 -911.458} C_VEL
LIN {X 0,Y 601.4,Z 270.198,A -85,B 0,C 180,E1 -912.358,E2 -912.358} C_VEL
LIN {X 0,Y 600.722,Z 270.281,A -85,B 0,C 180,E1 -912.918,E2 -912.918} C_VEL
LIN {X 0,Y 597.86,Z 270.642,A -85,B 0,C 180,E1 -913.826,E2 -913.826} C_VEL
LIN {X 0,Y 595.452,Z 270.941,A -85,B 0,C 180,E1 -914.556,E2 -914.556} C_VEL
LIN {X 0,Y 594.422,Z 271.068,A -85,B 0,C 180,E1 -915.119,E2 -915.119} C_VEL
LIN {X 0,Y 594.341,Z 271.076,A -85,B 0,C 180,E1 -915.31,E2 -915.31} C_VEL
LIN {X 0,Y 594.376,Z 271.071,A -85,B 0,C 180,E1 -917.904,E2 -917.904} C_VEL
LIN {X 0,Y 594.356,Z 271.073,A -85,B 0,C 180,E1 -920.913,E2 -920.913} C_VEL
LIN {X 0,Y 594.384,Z 271.069,A -85,B 0,C 180,E1 -923.704,E2 -923.704} C_VEL
LIN {X 0,Y 594.372,Z 271.071,A -85,B 0,C 180,E1 -926.7,E2 -926.7} C_VEL
LIN {X 0,Y 594.368,Z 271.071,A -85,B 0,C 180,E1 -929.777,E2 -929.777} C_VEL
LIN {X 0,Y 594.364,Z 271.078,A -85,B 0,C 180,E1 -932.147,E2 -932.147} C_VEL
LIN {X 0,Y 594.363,Z 271.072,A -85,B 0,C 180,E1 -934.581,E2 -934.581} C_VEL
LIN {X 0,Y 594.387,Z 271.069,A -85,B 0,C 180,E1 -937.61,E2 -937.61} C_VEL
LIN {X 0,Y 594.375,Z 271.077,A -85,B 0,C 180,E1 -939.776,E2 -939.776} C_VEL
LIN {X 0,Y 594.354,Z 271.074,A -85,B 0,C 180,E1 -942.377,E2 -942.377} C_VEL
LIN {X 0,Y 594.359,Z 271.073,A -85,B 0,C 180,E1 -945.192,E2 -945.192} C_VEL
LIN {X 0,Y 594.36,Z 271.077,A -85,B 0,C 180,E1 -947.625,E2 -947.625} C_VEL
LIN {X 0,Y 594.371,Z 271.074,A -85,B 0,C 180,E1 -948.536,E2 -948.536} C_VEL
LIN {X 0,Y 594.392,Z 275.669,A -85,B 0,C 180,E1 -951.295,E2 -951.295} C_VEL
LIN {X 0,Y 594.397,Z 279.967,A -85,B 0,C 180,E1 -953.76,E2 -953.76} C_VEL
LIN {X 0,Y 594.376,Z 284.419,A -85,B 0,C 180,E1 -956.24,E2 -956.24} C_VEL
LIN {X 0,Y 594.341,Z 288.831,A -85,B 0,C 180,E1 -958.649,E2 -958.649} C_VEL
LIN {X 0,Y 594.312,Z 294.773,A -85,B 0,C 180,E1 -961.77,E2 -961.77} C_VEL
LIN {X 0,Y 594.29,Z 300.737,A -85,B 0,C 180,E1 -964.804,E2 -964.804} C_VEL
LIN {X 0,Y 594.232,Z 306.702,A -85,B 0,C 180,E1 -967.762,E2 -967.762} C_VEL
LIN {X 0,Y 594.216,Z 311.176,A -85,B 0,C 180,E1 -969.941,E2 -969.941} C_VEL
LIN {X 0,Y 594.239,Z 317.141,A -85,B 0,C 180,E1 -972.803,E2 -972.803} C_VEL
LIN {X 0,Y 594.24,Z 317.807,A -85,B 0,C 180,E1 -973.094,E2 -973.094} C_VEL
LIN {X 0,Y 595.077,Z 322.394,A -85,B 0,C 180,E1 -973.184,E2 -973.184} C_VEL
LIN {X 0,Y 595.029,Z 337.716,A -85,B 0,C 180,E1 -973.48,E2 -973.48} C_VEL
LIN {X 0,Y 594.928,Z 353.196,A -85,B 0,C 180,E1 -973.927,E2 -973.927} C_VEL
LIN {X 0,Y 594.825,Z 367.794,A -85,B 0,C 180,E1 -974.496,E2 -974.496} C_VEL
LIN {X 0,Y 594.737,Z 381.873,A -85,B 0,C 180,E1 -975.195,E2 -975.195} C_VEL
LIN {X 0,Y 594.674,Z 394.639,A -85,B 0,C 180,E1 -975.973,E2 -975.973} C_VEL
LIN {X 0,Y 594.553,Z 407.684,A -85,B 0,C 180,E1 -976.935,E2 -976.935} C_VEL
LIN {X 0,Y 594.49,Z 418.515,A -85,B 0,C 180,E1 -977.888,E2 -977.888} C_VEL
LIN {X 0,Y 594.438,Z 428.342,A -85,B 0,C 180,E1 -978.904,E2 -978.904} C_VEL
LIN {X 0,Y 594.368,Z 438.296,A -85,B 0,C 180,E1 -980.128,E2 -980.128} C_VEL
LIN {X 0,Y 594.341,Z 446.454,A -85,B 0,C 180,E1 -981.329,E2 -981.329} C_VEL
LIN {X 0,Y 594.287,Z 453.188,A -85,B 0,C 180,E1 -982.526,E2 -982.526} C_VEL
LIN {X 0,Y 594.279,Z 459.422,A -85,B 0,C 180,E1 -983.891,E2 -983.891} C_VEL
LIN {X 0,Y 594.23,Z 464.244,A -85,B 0,C 180,E1 -985.251,E2 -985.251} C_VEL
LIN {X 0,Y 594.256,Z 467.792,A -85,B 0,C 180,E1 -986.61,E2 -986.61} C_VEL
LIN {X 0,Y 594.241,Z 470.141,A -85,B 0,C 180,E1 -987.967,E2 -987.967} C_VEL
LIN {X 0,Y 594.235,Z 471.337,A -85,B 0,C 180,E1 -989.323,E2 -989.323} C_VEL
LIN {X 0,Y 594.236,Z 471.361,A -85,B 0,C 180,E1 -990.678,E2 -990.678} C_VEL
LIN {X 0,Y 594.242,Z 470.244,A -85,B 0,C 180,E1 -992.034,E2 -992.034} C_VEL
LIN {X 0,Y 594.258,Z 467.982,A -85,B 0,C 180,E1 -993.39,E2 -993.39} C_VEL
LIN {X 0,Y 594.231,Z 464.523,A -85,B 0,C 180,E1 -994.749,E2 -994.749} C_VEL
LIN {X 0,Y 594.279,Z 459.794,A -85,B 0,C 180,E1 -996.11,E2 -996.11} C_VEL
LIN {X 0,Y 594.288,Z 453.663,A -85,B 0,C 180,E1 -997.475,E2 -997.475} C_VEL
LIN {X 0,Y 594.332,Z 445.945,A -85,B 0,C 180,E1 -998.843,E2 -998.843} C_VEL
LIN {X 0,Y 594.387,Z 437.703,A -85,B 0,C 180,E1 -1000.044,E2 -1000.044} C_VEL
LIN {X 0,Y 594.41,Z 427.979,A -85,B 0,C 180,E1 -1001.229,E2 -1001.229} C_VEL
LIN {X 0,Y 594.496,Z 417.654,A -85,B 0,C 180,E1 -1002.286,E2 -1002.286} C_VEL
LIN {X 0,Y 594.578,Z 405.583,A -85,B 0,C 180,E1 -1003.326,E2 -1003.326} C_VEL
LIN {X 0,Y 594.684,Z 392.135,A -85,B 0,C 180,E1 -1004.285,E2 -1004.285} C_VEL
LIN {X 0,Y 594.76,Z 378.747,A -85,B 0,C 180,E1 -1005.068,E2 -1005.068} C_VEL
LIN {X 0,Y 594.864,Z 364.864,A -85,B 0,C 180,E1 -1005.723,E2 -1005.723} C_VEL
LIN {X 0,Y 594.979,Z 350.641,A -85,B 0,C 180,E1 -1006.248,E2 -1006.248} C_VEL
LIN {X 0,Y 595.043,Z 335.667,A -85,B 0,C 180,E1 -1006.659,E2 -1006.659} C_VEL
LIN {X 0,Y 594.89,Z 320.853,A -85,B 0,C 180,E1 -1006.934,E2 -1006.934} C_VEL
LIN {X 0,Y 594.252,Z 317.711,A -85,B 0,C 180,E1 -1007.016,E2 -1007.016} C_VEL
LIN {X 0,Y 594.234,Z 312.853,A -85,B 0,C 180,E1 -1009.339,E2 -1009.339} C_VEL
LIN {X 0,Y 594.255,Z 308.376,A -85,B 0,C 180,E1 -1011.507,E2 -1011.507} C_VEL
LIN {X 0,Y 594.264,Z 302.408,A -85,B 0,C 180,E1 -1014.451,E2 -1014.451} C_VEL
LIN {X 0,Y 594.286,Z 297.931,A -85,B 0,C 180,E1 -1016.704,E2 -1016.704} C_VEL
LIN {X 0,Y 594.297,Z 293.454,A -85,B 0,C 180,E1 -1019.003,E2 -1019.003} C_VEL
LIN {X 0,Y 594.361,Z 288.471,A -85,B 0,C 180,E1 -1021.64,E2 -1021.64} C_VEL
LIN {X 0,Y 594.398,Z 283.097,A -85,B 0,C 180,E1 -1024.578,E2 -1024.578} C_VEL
LIN {X 0,Y 594.389,Z 278.632,A -85,B 0,C 180,E1 -1027.086,E2 -1027.086} C_VEL
LIN {X 0,Y 594.394,Z 273.991,A -85,B 0,C 180,E1 -1029.776,E2 -1029.776} C_VEL
LIN {X 0,Y 594.371,Z 271.175,A -85,B 0,C 180,E1 -1031.464,E2 -1031.464} C_VEL
LIN {X 0,Y 594.376,Z 271.076,A -85,B 0,C 180,E1 -1034.236,E2 -1034.236} C_VEL
LIN {X 0,Y 594.363,Z 271.073,A -85,B 0,C 180,E1 -1036.7,E2 -1036.7} C_VEL
LIN {X 0,Y 594.357,Z 271.073,A -85,B 0,C 180,E1 -1039.432,E2 -1039.432} C_VEL
LIN {X 0,Y 594.388,Z 271.072,A -85,B 0,C 180,E1 -1042.059,E2 -1042.059} C_VEL
LIN {X 0,Y 594.323,Z 271.081,A -85,B 0,C 180,E1 -1044.68,E2 -1044.68} C_VEL
LIN {X 0,Y 594.374,Z 271.071,A -85,B 0,C 180,E1 -1047.088,E2 -1047.088} C_VEL
LIN {X 0,Y 594.384,Z 271.073,A -85,B 0,C 180,E1 -1049.671,E2 -1049.671} C_VEL
LIN {X 0,Y 594.371,Z 271.077,A -85,B 0,C 180,E1 -1052.539,E2 -1052.539} C_VEL
LIN {X 0,Y 594.395,Z 271.074,A -85,B 0,C 180,E1 -1055.564,E2 -1055.564} C_VEL
LIN {X 0,Y 594.355,Z 271.077,A -85,B 0,C 180,E1 -1058.496,E2 -1058.496} C_VEL
LIN {X 0,Y 594.377,Z 271.072,A -85,B 0,C 180,E1 -1061.382,E2 -1061.382} C_VEL
LIN {X 0,Y 594.364,Z 271.072,A -85,B 0,C 180,E1 -1064.219,E2 -1064.219} C_VEL
LIN {X 0,Y 594.344,Z 271.074,A -85,B 0,C 180,E1 -1067.016,E2 -1067.016} C_VEL
LIN {X 0,Y 594.396,Z 271.069,A -85,B 0,C 180,E1 -1069.784,E2 -1069.784} C_VEL
LIN {X 0,Y 594.364,Z 271.076,A -85,B 0,C 180,E1 -1072.526,E2 -1072.526} C_VEL
LIN {X 0,Y 594.393,Z 271.072,A -85,B 0,C 180,E1 -1075.252,E2 -1075.252} C_VEL
LIN {X 0,Y 594.405,Z 271.067,A -85,B 0,C 180,E1 -1077.967,E2 -1077.967} C_VEL
LIN {X 0,Y 594.394,Z 271.068,A -85,B 0,C 180,E1 -1080.677,E2 -1080.677} C_VEL
LIN {X 0,Y 594.385,Z 271.072,A -85,B 0,C 180,E1 -1083.389,E2 -1083.389} C_VEL
LIN {X 0,Y 594.381,Z 271.075,A -85,B 0,C 180,E1 -1086.109,E2 -1086.109} C_VEL
LIN {X 0,Y 594.37,Z 271.073,A -85,B 0,C 180,E1 -1088.842,E2 -1088.842} C_VEL
LIN {X 0,Y 594.39,Z 271.069,A -85,B 0,C 180,E1 -1091.596,E2 -1091.596} C_VEL
LIN {X 0,Y 594.376,Z 271.071,A -85,B 0,C 180,E1 -1094.377,E2 -1094.377} C_VEL
LIN {X 0,Y 594.387,Z 271.071,A -85,B 0,C 180,E1 -1097.193,E2 -1097.193} C_VEL
LIN {X 0,Y 594.361,Z 271.077,A -85,B 0,C 180,E1 -1100.054,E2 -1100.054} C_VEL
LIN {X 0,Y 594.358,Z 271.079,A -85,B 0,C 180,E1 -1102.967,E2 -1102.967} C_VEL
LIN {X 0,Y 594.376,Z 271.07,A -85,B 0,C 180,E1 -1105.193,E2 -1105.193} C_VEL
LIN {X 0,Y 594.363,Z 271.078,A -85,B 0,C 180,E1 -1107.523,E2 -1107.523} C_VEL
LIN {X 0,Y 594.369,Z 271.074,A -85,B 0,C 180,E1 -1110.326,E2 -1110.326} C_VEL
LIN {X 0,Y 594.375,Z 271.071,A -85,B 0,C 180,E1 -1112.95,E2 -1112.95} C_VEL
LIN {X 0,Y 594.319,Z 271.082,A -85,B 0,C 180,E1 -1115.411,E2 -1115.411} C_VEL
LIN {X 0,Y 594.385,Z 271.072,A -85,B 0,C 180,E1 -1117.941,E2 -1117.941} C_VEL
LIN {X 0,Y 594.373,Z 271.072,A -85,B 0,C 180,E1 -1120.822,E2 -1120.822} C_VEL
LIN {X 0,Y 594.364,Z 271.073,A -85,B 0,C 180,E1 -1123.84,E2 -1123.84} C_VEL
LIN {X 0,Y 594.365,Z 271.073,A -85,B 0,C 180,E1 -1126.701,E2 -1126.701} C_VEL
LIN {X 0,Y 594.402,Z 271.227,A -85,B 0,C 180,E1 -1128.443,E2 -1128.443} C_VEL
LIN {X 0,Y 594.45,Z 274.953,A -85,B 0,C 180,E1 -1130.326,E2 -1130.326} C_VEL
LIN {X 0,Y 594.425,Z 280.256,A -85,B 0,C 180,E1 -1132.917,E2 -1132.917} C_VEL
LIN {X 0,Y 594.405,Z 285.597,A -85,B 0,C 180,E1 -1135.422,E2 -1135.422} C_VEL
LIN {X 0,Y 594.379,Z 290.967,A -85,B 0,C 180,E1 -1137.854,E2 -1137.854} C_VEL
LIN {X 0,Y 594.352,Z 296.32,A -85,B 0,C 180,E1 -1140.223,E2 -1140.223} C_VEL
LIN {X 0,Y 594.338,Z 301.638,A -85,B 0,C 180,E1 -1142.537,E2 -1142.537} C_VEL
LIN {X 0,Y 594.295,Z 306.957,A -85,B 0,C 180,E1 -1144.803,E2 -1144.803} C_VEL
LIN {X 0,Y 594.284,Z 314.048,A -85,B 0,C 180,E1 -1147.764,E2 -1147.764} C_VEL
LIN {X 0,Y 594.276,Z 321.139,A -85,B 0,C 180,E1 -1150.663,E2 -1150.663} C_VEL
LIN {X 0,Y 594.251,Z 327.05,A -85,B 0,C 180,E1 -1153.04,E2 -1153.04} C_VEL
LIN {X 0,Y 595.086,Z 331.585,A -85,B 0,C 180,E1 -1153.127,E2 -1153.127} C_VEL
LIN {X 0,Y 595.023,Z 347.061,A -85,B 0,C 180,E1 -1153.419,E2 -1153.419} C_VEL
LIN {X 0,Y 594.952,Z 361.911,A -85,B 0,C 180,E1 -1153.839,E2 -1153.839} C_VEL
LIN {X 0,Y 594.863,Z 374.84,A -85,B 0,C 180,E1 -1154.32,E2 -1154.32} C_VEL
LIN {X 0,Y 594.761,Z 389.526,A -85,B 0,C 180,E1 -1155.02,E2 -1155.02} C_VEL
LIN {X 0,Y 594.673,Z 403.073,A -85,B 0,C 180,E1 -1155.822,E2 -1155.822} C_VEL
LIN {X 0,Y 594.596,Z 416.099,A -85,B 0,C 180,E1 -1156.761,E2 -1156.761} C_VEL
LIN {X 0,Y 594.53,Z 427.19,A -85,B 0,C 180,E1 -1157.715,E2 -1157.715} C_VEL
LIN {X 0,Y 594.455,Z 437.281,A -85,B 0,C 180,E1 -1158.739,E2 -1158.739} C_VEL
LIN {X 0,Y 594.387,Z 447.369,A -85,B 0,C 180,E1 -1159.956,E2 -1159.956} C_VEL
LIN {X 0,Y 594.331,Z 455.652,A -85,B 0,C 180,E1 -1161.157,E2 -1161.157} C_VEL
LIN {X 0,Y 594.287,Z 463.425,A -85,B 0,C 180,E1 -1162.525,E2 -1162.525} C_VEL
LIN {X 0,Y 594.279,Z 469.607,A -85,B 0,C 180,E1 -1163.89,E2 -1163.89} C_VEL
LIN {X 0,Y 594.232,Z 474.383,A -85,B 0,C 180,E1 -1165.251,E2 -1165.251} C_VEL
LIN {X 0,Y 594.257,Z 477.886,A -85,B 0,C 180,E1 -1166.61,E2 -1166.61} C_VEL
LIN {X 0,Y 594.241,Z 480.192,A -85,B 0,C 180,E1 -1167.966,E2 -1167.966} C_VEL
LIN {X 0,Y 594.235,Z 481.35,A -85,B 0,C 180,E1 -1169.322,E2 -1169.322} C_VEL
LIN {X 0,Y 594.235,Z 481.35,A -85,B 0,C 180,E1 -1170.677,E2 -1170.677} C_VEL
LIN {X 0,Y 594.241,Z 480.193,A -85,B 0,C 180,E1 -1172.033,E2 -1172.033} C_VEL
LIN {X 0,Y 594.257,Z 477.887,A -85,B 0,C 180,E1 -1173.39,E2 -1173.39} C_VEL
LIN {X 0,Y 594.232,Z 474.385,A -85,B 0,C 180,E1 -1174.749,E2 -1174.749} C_VEL
LIN {X 0,Y 594.279,Z 469.609,A -85,B 0,C 180,E1 -1176.109,E2 -1176.109} C_VEL
LIN {X 0,Y 594.286,Z 463.427,A -85,B 0,C 180,E1 -1177.474,E2 -1177.474} C_VEL
LIN {X 0,Y 594.331,Z 455.655,A -85,B 0,C 180,E1 -1178.842,E2 -1178.842} C_VEL
LIN {X 0,Y 594.387,Z 447.373,A -85,B 0,C 180,E1 -1180.044,E2 -1180.044} C_VEL
LIN {X 0,Y 594.433,Z 437.562,A -85,B 0,C 180,E1 -1181.231,E2 -1181.231} C_VEL
LIN {X 0,Y 594.53,Z 427.196,A -85,B 0,C 180,E1 -1182.285,E2 -1182.285} C_VEL
LIN {X 0,Y 594.581,Z 415.023,A -85,B 0,C 180,E1 -1183.326,E2 -1183.326} C_VEL
LIN {X 0,Y 594.693,Z 403.082,A -85,B 0,C 180,E1 -1184.177,E2 -1184.177} C_VEL
LIN {X 0,Y 594.76,Z 389.534,A -85,B 0,C 180,E1 -1184.98,E2 -1184.98} C_VEL
LIN {X 0,Y 594.865,Z 374.852,A -85,B 0,C 180,E1 -1185.679,E2 -1185.679} C_VEL
LIN {X 0,Y 594.957,Z 360.633,A -85,B 0,C 180,E1 -1186.204,E2 -1186.204} C_VEL
LIN {X 0,Y 595.044,Z 345.927,A -85,B 0,C 180,E1 -1186.608,E2 -1186.608} C_VEL
LIN {X 0,Y 594.945,Z 330.358,A -85,B 0,C 180,E1 -1186.895,E2 -1186.895} C_VEL
LIN {X 0,Y 594.245,Z 327.008,A -85,B 0,C 180,E1 -1186.978,E2 -1186.978} C_VEL
LIN {X 0,Y 594.275,Z 321.14,A -85,B 0,C 180,E1 -1189.337,E2 -1189.337} C_VEL
LIN {X 0,Y 594.283,Z 314.049,A -85,B 0,C 180,E1 -1192.236,E2 -1192.236} C_VEL
LIN {X 0,Y 594.296,Z 306.958,A -85,B 0,C 180,E1 -1195.196,E2 -1195.196} C_VEL
LIN {X 0,Y 594.338,Z 301.51,A -85,B 0,C 180,E1 -1197.518,E2 -1197.518} C_VEL
LIN {X 0,Y 594.364,Z 295.077,A -85,B 0,C 180,E1 -1200.325,E2 -1200.325} C_VEL
LIN {X 0,Y 594.422,Z 289.179,A -85,B 0,C 180,E1 -1202.947,E2 -1202.947} C_VEL
LIN {X 0,Y 594.443,Z 283.812,A -85,B 0,C 180,E1 -1205.402,E2 -1205.402} C_VEL
LIN {X 0,Y 594.451,Z 278.489,A -85,B 0,C 180,E1 -1207.935,E2 -1207.935} C_VEL
LIN {X 0,Y 594.504,Z 272.627,A -85,B 0,C 180,E1 -1210.836,E2 -1210.836} C_VEL
LIN {X 0,Y 594.372,Z 271.075,A -85,B 0,C 180,E1 -1211.655,E2 -1211.655} C_VEL
LIN {X 0,Y 594.376,Z 271.075,A -85,B 0,C 180,E1 -1214.236,E2 -1214.236} C_VEL
LIN {X 0,Y 594.351,Z 271.08,A -85,B 0,C 180,E1 -1217.148,E2 -1217.148} C_VEL
LIN {X 0,Y 594.359,Z 271.073,A -85,B 0,C 180,E1 -1219.432,E2 -1219.432} C_VEL
LIN {X 0,Y 594.384,Z 271.072,A -85,B 0,C 180,E1 -1222.059,E2 -1222.059} C_VEL
LIN {X 0,Y 594.319,Z 271.082,A -85,B 0,C 180,E1 -1224.679,E2 -1224.679} C_VEL
LIN {X 0,Y 594.372,Z 271.071,A -85,B 0,C 180,E1 -1227.088,E2 -1227.088} C_VEL
LIN {X 0,Y 594.379,Z 271.073,A -85,B 0,C 180,E1 -1229.671,E2 -1229.671} C_VEL
LIN {X 0,Y 594.366,Z 271.077,A -85,B 0,C 180,E1 -1232.539,E2 -1232.539} C_VEL
LIN {X 0,Y 594.374,Z 271.071,A -85,B 0,C 180,E1 -1234.807,E2 -1234.807} C_VEL
LIN {X 0,Y 594.357,Z 271.076,A -85,B 0,C 180,E1 -1237.264,E2 -1237.264} C_VEL
LIN {X 0,Y 594.358,Z 271.077,A -85,B 0,C 180,E1 -1239.946,E2 -1239.946} C_VEL
LIN {X 0,Y 594.385,Z 271.071,A -85,B 0,C 180,E1 -1242.807,E2 -1242.807} C_VEL
LIN {X 0,Y 594.376,Z 271.072,A -85,B 0,C 180,E1 -1245.827,E2 -1245.827} C_VEL
LIN {X 0,Y 594.387,Z 271.069,A -85,B 0,C 180,E1 -1248.404,E2 -1248.404} C_VEL
LIN {X 0,Y 594.37,Z 271.073,A -85,B 0,C 180,E1 -1251.158,E2 -1251.158} C_VEL
LIN {X 0,Y 594.38,Z 271.076,A -85,B 0,C 180,E1 -1253.891,E2 -1253.891} C_VEL
LIN {X 0,Y 594.383,Z 271.072,A -85,B 0,C 180,E1 -1256.611,E2 -1256.611} C_VEL
LIN {X 0,Y 594.392,Z 271.068,A -85,B 0,C 180,E1 -1259.323,E2 -1259.323} C_VEL
LIN {X 0,Y 594.404,Z 271.068,A -85,B 0,C 180,E1 -1262.033,E2 -1262.033} C_VEL
LIN {X 0,Y 594.394,Z 271.072,A -85,B 0,C 180,E1 -1264.748,E2 -1264.748} C_VEL
LIN {X 0,Y 594.36,Z 271.076,A -85,B 0,C 180,E1 -1267.474,E2 -1267.474} C_VEL
LIN {X 0,Y 594.394,Z 271.069,A -85,B 0,C 180,E1 -1270.216,E2 -1270.216} C_VEL
LIN {X 0,Y 594.348,Z 271.074,A -85,B 0,C 180,E1 -1272.984,E2 -1272.984} C_VEL
LIN {X 0,Y 594.341,Z 271.076,A -85,B 0,C 180,E1 -1275.31,E2 -1275.31} C_VEL
LIN {X 0,Y 593.682,Z 271.158,A -85,B 0,C 180,E1 -1275.876,E2 -1275.876} C_VEL
LIN {X 0,Y 590.837,Z 271.517,A -85,B 0,C 180,E1 -1276.794,E2 -1276.794} C_VEL
LIN {X 0,Y 588.431,Z 271.816,A -85,B 0,C 180,E1 -1277.533,E2 -1277.533} C_VEL
LIN {X 0,Y 587.401,Z 271.942,A -85,B 0,C 180,E1 -1278.103,E2 -1278.103} C_VEL
LIN {X 0,Y 587.318,Z 271.951,A -85,B 0,C 180,E1 -1278.296,E2 -1278.296} C_VEL
LIN {X 0,Y 587.322,Z 271.951,A -85,B 0,C 180,E1 -1281.038,E2 -1281.038} C_VEL
LIN {X 0,Y 587.316,Z 271.952,A -85,B 0,C 180,E1 -1283.259,E2 -1283.259} C_VEL
LIN {X 0,Y 587.332,Z 271.949,A -85,B 0,C 180,E1 -1285.517,E2 -1285.517} C_VEL
LIN {X 0,Y 587.328,Z 271.951,A -85,B 0,C 180,E1 -1287.819,E2 -1287.819} C_VEL
LIN {X 0,Y 587.335,Z 271.952,A -85,B 0,C 180,E1 -1290.511,E2 -1290.511} C_VEL
LIN {X 0,Y 587.333,Z 271.948,A -85,B 0,C 180,E1 -1293.113,E2 -1293.113} C_VEL
LIN {X 0,Y 587.269,Z 271.957,A -85,B 0,C 180,E1 -1295.535,E2 -1295.535} C_VEL
LIN {X 0,Y 587.338,Z 271.948,A -85,B 0,C 180,E1 -1297.84,E2 -1297.84} C_VEL
LIN {X 0,Y 587.311,Z 271.951,A -85,B 0,C 180,E1 -1300.255,E2 -1300.255} C_VEL
LIN {X 0,Y 587.308,Z 271.953,A -85,B 0,C 180,E1 -1303.119,E2 -1303.119} C_VEL
LIN {X 0,Y 587.331,Z 271.953,A -85,B 0,C 180,E1 -1306.051,E2 -1306.051} C_VEL
LIN {X 0,Y 587.314,Z 271.953,A -85,B 0,C 180,E1 -1307.925,E2 -1307.925} C_VEL
LIN {X 0,Y 587.359,Z 272.665,A -85,B 0,C 180,E1 -1308.923,E2 -1308.923} C_VEL
LIN {X 0,Y 587.342,Z 277.005,A -85,B 0,C 180,E1 -1311.523,E2 -1311.523} C_VEL
LIN {X 0,Y 587.352,Z 282.086,A -85,B 0,C 180,E1 -1314.455,E2 -1314.455} C_VEL
LIN {X 0,Y 587.335,Z 286.445,A -85,B 0,C 180,E1 -1316.889,E2 -1316.889} C_VEL
LIN {X 0,Y 587.246,Z 291.219,A -85,B 0,C 180,E1 -1319.505,E2 -1319.505} C_VEL
LIN {X 0,Y 587.27,Z 296.542,A -85,B 0,C 180,E1 -1322.323,E2 -1322.323} C_VEL
LIN {X 0,Y 587.214,Z 302.23,A -85,B 0,C 180,E1 -1325.236,E2 -1325.236} C_VEL
LIN {X 0,Y 587.17,Z 306.703,A -85,B 0,C 180,E1 -1327.48,E2 -1327.48} C_VEL
LIN {X 0,Y 587.149,Z 311.177,A -85,B 0,C 180,E1 -1329.689,E2 -1329.689} C_VEL
LIN {X 0,Y 587.174,Z 317.142,A -85,B 0,C 180,E1 -1332.589,E2 -1332.589} C_VEL
LIN {X 0,Y 587.169,Z 317.899,A -85,B 0,C 180,E1 -1332.884,E2 -1332.884} C_VEL
LIN {X 0,Y 588.318,Z 323.751,A -85,B 0,C 180,E1 -1333.004,E2 -1333.004} C_VEL
LIN {X 0,Y 588.234,Z 339.034,A -85,B 0,C 180,E1 -1333.315,E2 -1333.315} C_VEL
LIN {X 0,Y 588.071,Z 354.507,A -85,B 0,C 180,E1 -1333.779,E2 -1333.779} C_VEL
LIN {X 0,Y 587.952,Z 367.808,A -85,B 0,C 180,E1 -1334.31,E2 -1334.31} C_VEL
LIN {X 0,Y 587.828,Z 381.885,A -85,B 0,C 180,E1 -1335.017,E2 -1335.017} C_VEL
LIN {X 0,Y 587.721,Z 395.194,A -85,B 0,C 180,E1 -1335.841,E2 -1335.841} C_VEL
LIN {X 0,Y 587.569,Z 407.693,A -85,B 0,C 180,E1 -1336.777,E2 -1336.777} C_VEL
LIN {X 0,Y 587.503,Z 418.52,A -85,B 0,C 180,E1 -1337.741,E2 -1337.741} C_VEL
LIN {X 0,Y 587.394,Z 428.995,A -85,B 0,C 180,E1 -1338.845,E2 -1338.845} C_VEL
LIN {X 0,Y 587.334,Z 438.301,A -85,B 0,C 180,E1 -1340.009,E2 -1340.009} C_VEL
LIN {X 0,Y 587.269,Z 446.458,A -85,B 0,C 180,E1 -1341.224,E2 -1341.224} C_VEL
LIN {X 0,Y 587.23,Z 453.191,A -85,B 0,C 180,E1 -1342.436,E2 -1342.436} C_VEL
LIN {X 0,Y 587.18,Z 459.424,A -85,B 0,C 180,E1 -1343.816,E2 -1343.816} C_VEL
LIN {X 0,Y 587.134,Z 464.247,A -85,B 0,C 180,E1 -1345.194,E2 -1345.194} C_VEL
LIN {X 0,Y 587.179,Z 467.793,A -85,B 0,C 180,E1 -1346.569,E2 -1346.569} C_VEL
LIN {X 0,Y 587.14,Z 470.141,A -85,B 0,C 180,E1 -1347.942,E2 -1347.942} C_VEL
LIN {X 0,Y 587.135,Z 471.337,A -85,B 0,C 180,E1 -1349.314,E2 -1349.314} C_VEL
LIN {X 0,Y 587.136,Z 471.36,A -85,B 0,C 180,E1 -1350.686,E2 -1350.686} C_VEL
LIN {X 0,Y 587.14,Z 470.244,A -85,B 0,C 180,E1 -1352.058,E2 -1352.058} C_VEL
LIN {X 0,Y 587.181,Z 467.981,A -85,B 0,C 180,E1 -1353.431,E2 -1353.431} C_VEL
LIN {X 0,Y 587.134,Z 464.522,A -85,B 0,C 180,E1 -1354.807,E2 -1354.807} C_VEL
LIN {X 0,Y 587.183,Z 459.792,A -85,B 0,C 180,E1 -1356.184,E2 -1356.184} C_VEL
LIN {X 0,Y 587.231,Z 453.66,A -85,B 0,C 180,E1 -1357.565,E2 -1357.565} C_VEL
LIN {X 0,Y 587.266,Z 445.941,A -85,B 0,C 180,E1 -1358.95,E2 -1358.95} C_VEL
LIN {X 0,Y 587.351,Z 437.699,A -85,B 0,C 180,E1 -1360.166,E2 -1360.166} C_VEL
LIN {X 0,Y 587.398,Z 427.795,A -85,B 0,C 180,E1 -1361.386,E2 -1361.386} C_VEL
LIN {X 0,Y 587.492,Z 417.647,A -85,B 0,C 180,E1 -1362.435,E2 -1362.435} C_VEL
LIN {X 0,Y 587.621,Z 405.574,A -85,B 0,C 180,E1 -1363.487,E2 -1363.487} C_VEL
LIN {X 0,Y 587.775,Z 391.92,A -85,B 0,C 180,E1 -1364.47,E2 -1364.47} C_VEL
LIN {X 0,Y 587.863,Z 378.737,A -85,B 0,C 180,E1 -1365.249,E2 -1365.249} C_VEL
LIN {X 0,Y 588.015,Z 364.849,A -85,B 0,C 180,E1 -1365.911,E2 -1365.911} C_VEL
LIN {X 0,Y 588.156,Z 350.622,A -85,B 0,C 180,E1 -1366.442,E2 -1366.442} C_VEL
LIN {X 0,Y 588.239,Z 335.359,A -85,B 0,C 180,E1 -1366.864,E2 -1366.864} C_VEL
LIN {X 0,Y 588.083,Z 321.913,A -85,B 0,C 180,E1 -1367.12,E2 -1367.12} C_VEL
LIN {X 0,Y 587.156,Z 317.72,A -85,B 0,C 180,E1 -1367.223,E2 -1367.223} C_VEL
LIN {X 0,Y 587.164,Z 312.852,A -85,B 0,C 180,E1 -1369.581,E2 -1369.581} C_VEL
LIN {X 0,Y 587.158,Z 308.375,A -85,B 0,C 180,E1 -1371.781,E2 -1371.781} C_VEL
LIN {X 0,Y 587.188,Z 302.844,A -85,B 0,C 180,E1 -1374.545,E2 -1374.545} C_VEL
LIN {X 0,Y 587.226,Z 297.93,A -85,B 0,C 180,E1 -1377.051,E2 -1377.051} C_VEL
LIN {X 0,Y 587.225,Z 293.465,A -85,B 0,C 180,E1 -1379.386,E2 -1379.386} C_VEL
LIN {X 0,Y 587.313,Z 288.934,A -85,B 0,C 180,E1 -1381.83,E2 -1381.83} C_VEL
LIN {X 0,Y 587.357,Z 284.375,A -85,B 0,C 180,E1 -1384.349,E2 -1384.349} C_VEL
LIN {X 0,Y 587.355,Z 280.147,A -85,B 0,C 180,E1 -1386.746,E2 -1386.746} C_VEL
LIN {X 0,Y 587.351,Z 275.668,A -85,B 0,C 180,E1 -1389.358,E2 -1389.358} C_VEL
LIN {X 0,Y 587.359,Z 272.688,A -85,B 0,C 180,E1 -1391.155,E2 -1391.155} C_VEL
LIN {X 0,Y 587.334,Z 271.951,A -85,B 0,C 180,E1 -1392.107,E2 -1392.107} C_VEL
LIN {X 0,Y 587.315,Z 271.951,A -85,B 0,C 180,E1 -1395.088,E2 -1395.088} C_VEL
LIN {X 0,Y 587.311,Z 271.951,A -85,B 0,C 180,E1 -1397.924,E2 -1397.924} C_VEL
LIN {X 0,Y 587.347,Z 271.948,A -85,B 0,C 180,E1 -1400.641,E2 -1400.641} C_VEL
LIN {X 0,Y 587.346,Z 271.952,A -85,B 0,C 180,E1 -1403.292,E2 -1403.292} C_VEL
LIN {X 0,Y 587.349,Z 271.946,A -85,B 0,C 180,E1 -1405.779,E2 -1405.779} C_VEL
LIN {X 0,Y 587.348,Z 271.948,A -85,B 0,C 180,E1 -1408.231,E2 -1408.231} C_VEL
LIN {X 0,Y 587.343,Z 271.951,A -85,B 0,C 180,E1 -1410.867,E2 -1410.867} C_VEL
LIN {X 0,Y 587.326,Z 271.951,A -85,B 0,C 180,E1 -1413.824,E2 -1413.824} C_VEL
LIN {X 0,Y 587.335,Z 271.949,A -85,B 0,C 180,E1 -1415.993,E2 -1415.993} C_VEL
LIN {X 0,Y 587.311,Z 271.951,A -85,B 0,C 180,E1 -1418.225,E2 -1418.225} C_VEL
LIN {X 0,Y 587.341,Z 271.947,A -85,B 0,C 180,E1 -1421.151,E2 -1421.151} C_VEL
LIN {X 0,Y 587.345,Z 271.951,A -85,B 0,C 180,E1 -1423.311,E2 -1423.311} C_VEL
LIN {X 0,Y 587.339,Z 271.951,A -85,B 0,C 180,E1 -1426.154,E2 -1426.154} C_VEL
LIN {X 0,Y 587.34,Z 271.948,A -85,B 0,C 180,E1 -1428.962,E2 -1428.962} C_VEL
LIN {X 0,Y 587.359,Z 271.944,A -85,B 0,C 180,E1 -1431.745,E2 -1431.745} C_VEL
LIN {X 0,Y 587.348,Z 271.946,A -85,B 0,C 180,E1 -1434.507,E2 -1434.507} C_VEL
LIN {X 0,Y 587.367,Z 271.946,A -85,B 0,C 180,E1 -1437.257,E2 -1437.257} C_VEL
LIN {X 0,Y 587.378,Z 271.948,A -85,B 0,C 180,E1 -1440,E2 -1440} C_VEL
LIN {X 0,Y 587.365,Z 271.945,A -85,B 0,C 180,E1 -1442.743,E2 -1442.743} C_VEL
LIN {X 0,Y 587.351,Z 271.945,A -85,B 0,C 180,E1 -1445.493,E2 -1445.493} C_VEL
LIN {X 0,Y 587.358,Z 271.945,A -85,B 0,C 180,E1 -1448.255,E2 -1448.255} C_VEL
LIN {X 0,Y 587.343,Z 271.948,A -85,B 0,C 180,E1 -1451.134,E2 -1451.134} C_VEL
LIN {X 0,Y 587.349,Z 271.952,A -85,B 0,C 180,E1 -1453.846,E2 -1453.846} C_VEL
LIN {X 0,Y 587.352,Z 271.951,A -85,B 0,C 180,E1 -1456.817,E2 -1456.817} C_VEL
LIN {X 0,Y 587.306,Z 271.953,A -85,B 0,C 180,E1 -1459.576,E2 -1459.576} C_VEL
LIN {X 0,Y 587.309,Z 271.953,A -85,B 0,C 180,E1 -1461.775,E2 -1461.775} C_VEL
LIN {X 0,Y 587.349,Z 271.949,A -85,B 0,C 180,E1 -1464.759,E2 -1464.759} C_VEL
LIN {X 0,Y 587.322,Z 271.95,A -85,B 0,C 180,E1 -1467.046,E2 -1467.046} C_VEL
LIN {X 0,Y 587.309,Z 271.954,A -85,B 0,C 180,E1 -1469.382,E2 -1469.382} C_VEL
LIN {X 0,Y 587.352,Z 271.948,A -85,B 0,C 180,E1 -1471.838,E2 -1471.838} C_VEL
LIN {X 0,Y 587.335,Z 271.948,A -85,B 0,C 180,E1 -1474.347,E2 -1474.347} C_VEL
LIN {X 0,Y 587.344,Z 271.947,A -85,B 0,C 180,E1 -1477.608,E2 -1477.608} C_VEL
LIN {X 0,Y 587.313,Z 271.951,A -85,B 0,C 180,E1 -1480.254,E2 -1480.254} C_VEL
LIN {X 0,Y 587.309,Z 271.954,A -85,B 0,C 180,E1 -1483.118,E2 -1483.118} C_VEL
LIN {X 0,Y 587.322,Z 271.955,A -85,B 0,C 180,E1 -1486.05,E2 -1486.05} C_VEL
LIN {X 0,Y 587.344,Z 272.061,A -85,B 0,C 180,E1 -1488.273,E2 -1488.273} C_VEL
LIN {X 0,Y 587.458,Z 275.346,A -85,B 0,C 180,E1 -1489.965,E2 -1489.965} C_VEL
LIN {X 0,Y 587.409,Z 280.249,A -85,B 0,C 180,E1 -1492.398,E2 -1492.398} C_VEL
LIN {X 0,Y 587.389,Z 285.564,A -85,B 0,C 180,E1 -1494.949,E2 -1494.949} C_VEL
LIN {X 0,Y 587.367,Z 290.93,A -85,B 0,C 180,E1 -1497.423,E2 -1497.423} C_VEL
LIN {X 0,Y 587.308,Z 296.295,A -85,B 0,C 180,E1 -1499.829,E2 -1499.829} C_VEL
LIN {X 0,Y 587.294,Z 301.954,A -85,B 0,C 180,E1 -1502.318,E2 -1502.318} C_VEL
LIN {X 0,Y 587.22,Z 308.73,A -85,B 0,C 180,E1 -1505.236,E2 -1505.236} C_VEL
LIN {X 0,Y 587.235,Z 314.048,A -85,B 0,C 180,E1 -1507.482,E2 -1507.482} C_VEL
LIN {X 0,Y 587.199,Z 321.139,A -85,B 0,C 180,E1 -1510.42,E2 -1510.42} C_VEL
LIN {X 0,Y 587.19,Z 327.047,A -85,B 0,C 180,E1 -1512.828,E2 -1512.828} C_VEL
LIN {X 0,Y 588.309,Z 332.76,A -85,B 0,C 180,E1 -1512.944,E2 -1512.944} C_VEL
LIN {X 0,Y 588.216,Z 348.067,A -85,B 0,C 180,E1 -1513.246,E2 -1513.246} C_VEL
LIN {X 0,Y 588.113,Z 363.206,A -85,B 0,C 180,E1 -1513.69,E2 -1513.69} C_VEL
LIN {X 0,Y 587.984,Z 376.825,A -85,B 0,C 180,E1 -1514.221,E2 -1514.221} C_VEL
LIN {X 0,Y 587.863,Z 391.104,A -85,B 0,C 180,E1 -1514.928,E2 -1514.928} C_VEL
LIN {X 0,Y 587.726,Z 404.571,A -85,B 0,C 180,E1 -1515.753,E2 -1515.753} C_VEL
LIN {X 0,Y 587.616,Z 417.166,A -85,B 0,C 180,E1 -1516.689,E2 -1516.689} C_VEL
LIN {X 0,Y 587.503,Z 428.972,A -85,B 0,C 180,E1 -1517.741,E2 -1517.741} C_VEL
LIN {X 0,Y 587.361,Z 439.517,A -85,B 0,C 180,E1 -1518.86,E2 -1518.86} C_VEL
LIN {X 0,Y 587.334,Z 448.617,A -85,B 0,C 180,E1 -1520.008,E2 -1520.008} C_VEL
LIN {X 0,Y 587.27,Z 456.719,A -85,B 0,C 180,E1 -1521.223,E2 -1521.223} C_VEL
LIN {X 0,Y 587.23,Z 463.425,A -85,B 0,C 180,E1 -1522.435,E2 -1522.435} C_VEL
LIN {X 0,Y 587.18,Z 469.606,A -85,B 0,C 180,E1 -1523.816,E2 -1523.816} C_VEL
LIN {X 0,Y 587.136,Z 474.383,A -85,B 0,C 180,E1 -1525.193,E2 -1525.193} C_VEL
LIN {X 0,Y 587.18,Z 477.887,A -85,B 0,C 180,E1 -1526.569,E2 -1526.569} C_VEL
LIN {X 0,Y 587.14,Z 480.193,A -85,B 0,C 180,E1 -1527.942,E2 -1527.942} C_VEL
LIN {X 0,Y 587.135,Z 481.35,A -85,B 0,C 180,E1 -1529.314,E2 -1529.314} C_VEL
LIN {X 0,Y 587.135,Z 481.35,A -85,B 0,C 180,E1 -1530.686,E2 -1530.686} C_VEL
LIN {X 0,Y 587.14,Z 480.193,A -85,B 0,C 180,E1 -1532.058,E2 -1532.058} C_VEL
LIN {X 0,Y 587.179,Z 477.887,A -85,B 0,C 180,E1 -1533.431,E2 -1533.431} C_VEL
LIN {X 0,Y 587.136,Z 474.385,A -85,B 0,C 180,E1 -1534.806,E2 -1534.806} C_VEL
LIN {X 0,Y 587.18,Z 469.61,A -85,B 0,C 180,E1 -1536.184,E2 -1536.184} C_VEL
LIN {X 0,Y 587.229,Z 463.426,A -85,B 0,C 180,E1 -1537.564,E2 -1537.564} C_VEL
LIN {X 0,Y 587.266,Z 455.654,A -85,B 0,C 180,E1 -1538.95,E2 -1538.95} C_VEL
LIN {X 0,Y 587.351,Z 447.373,A -85,B 0,C 180,E1 -1540.165,E2 -1540.165} C_VEL
LIN {X 0,Y 587.399,Z 437.399,A -85,B 0,C 180,E1 -1541.385,E2 -1541.385} C_VEL
LIN {X 0,Y 587.522,Z 427.196,A -85,B 0,C 180,E1 -1542.434,E2 -1542.434} C_VEL
LIN {X 0,Y 587.629,Z 415.024,A -85,B 0,C 180,E1 -1543.486,E2 -1543.486} C_VEL
LIN {X 0,Y 587.773,Z 402.063,A -85,B 0,C 180,E1 -1544.416,E2 -1544.416} C_VEL
LIN {X 0,Y 587.856,Z 387.875,A -85,B 0,C 180,E1 -1545.249,E2 -1545.249} C_VEL
LIN {X 0,Y 588.027,Z 373.808,A -85,B 0,C 180,E1 -1545.911,E2 -1545.911} C_VEL
LIN {X 0,Y 588.164,Z 359.319,A -85,B 0,C 180,E1 -1546.441,E2 -1546.441} C_VEL
LIN {X 0,Y 588.227,Z 344.084,A -85,B 0,C 180,E1 -1546.85,E2 -1546.85} C_VEL
LIN {X 0,Y 588.175,Z 331.512,A -85,B 0,C 180,E1 -1547.078,E2 -1547.078} C_VEL
LIN {X 0,Y 587.189,Z 327.047,A -85,B 0,C 180,E1 -1547.172,E2 -1547.172} C_VEL
LIN {X 0,Y 587.198,Z 321.14,A -85,B 0,C 180,E1 -1549.579,E2 -1549.579} C_VEL
LIN {X 0,Y 587.233,Z 314.049,A -85,B 0,C 180,E1 -1552.517,E2 -1552.517} C_VEL
LIN {X 0,Y 587.232,Z 306.958,A -85,B 0,C 180,E1 -1555.521,E2 -1555.521} C_VEL
LIN {X 0,Y 587.285,Z 301.64,A -85,B 0,C 180,E1 -1557.82,E2 -1557.82} C_VEL
LIN {X 0,Y 587.32,Z 295.538,A -85,B 0,C 180,E1 -1560.507,E2 -1560.507} C_VEL
LIN {X 0,Y 587.39,Z 289.738,A -85,B 0,C 180,E1 -1563.119,E2 -1563.119} C_VEL
LIN {X 0,Y 587.386,Z 283.787,A -85,B 0,C 180,E1 -1565.892,E2 -1565.892} C_VEL
LIN {X 0,Y 587.457,Z 278.486,A -85,B 0,C 180,E1 -1568.468,E2 -1568.468} C_VEL
LIN {X 0,Y 587.473,Z 273.167,A -85,B 0,C 180,E1 -1571.144,E2 -1571.144} C_VEL
LIN {X 0,Y 587.331,Z 271.953,A -85,B 0,C 180,E1 -1571.843,E2 -1571.843} C_VEL
LIN {X 0,Y 587.329,Z 271.953,A -85,B 0,C 180,E1 -1574.114,E2 -1574.114} C_VEL
LIN {X 0,Y 587.305,Z 271.956,A -85,B 0,C 180,E1 -1576.993,E2 -1576.993} C_VEL
LIN {X 0,Y 587.311,Z 271.952,A -85,B 0,C 180,E1 -1579.745,E2 -1579.745} C_VEL
LIN {X 0,Y 587.341,Z 271.947,A -85,B 0,C 180,E1 -1582.392,E2 -1582.392} C_VEL
LIN {X 0,Y 587.347,Z 271.947,A -85,B 0,C 180,E1 -1585.779,E2 -1585.779} C_VEL
LIN {X 0,Y 587.347,Z 271.948,A -85,B 0,C 180,E1 -1588.232,E2 -1588.232} C_VEL
LIN {X 0,Y 587.338,Z 271.953,A -85,B 0,C 180,E1 -1590.867,E2 -1590.867} C_VEL
LIN {X 0,Y 587.353,Z 271.949,A -85,B 0,C 180,E1 -1593.818,E2 -1593.818} C_VEL
LIN {X 0,Y 587.33,Z 271.949,A -85,B 0,C 180,E1 -1595.993,E2 -1595.993} C_VEL
LIN {X 0,Y 587.307,Z 271.953,A -85,B 0,C 180,E1 -1598.225,E2 -1598.225} C_VEL
LIN {X 0,Y 587.341,Z 271.947,A -85,B 0,C 180,E1 -1601.151,E2 -1601.151} C_VEL
LIN {X 0,Y 587.34,Z 271.951,A -85,B 0,C 180,E1 -1603.311,E2 -1603.311} C_VEL
LIN {X 0,Y 587.345,Z 271.951,A -85,B 0,C 180,E1 -1606.154,E2 -1606.154} C_VEL
LIN {X 0,Y 587.338,Z 271.949,A -85,B 0,C 180,E1 -1608.962,E2 -1608.962} C_VEL
LIN {X 0,Y 587.356,Z 271.945,A -85,B 0,C 180,E1 -1611.745,E2 -1611.745} C_VEL
LIN {X 0,Y 587.349,Z 271.946,A -85,B 0,C 180,E1 -1614.507,E2 -1614.507} C_VEL
LIN {X 0,Y 587.365,Z 271.945,A -85,B 0,C 180,E1 -1617.257,E2 -1617.257} C_VEL
LIN {X 0,Y 587.375,Z 271.949,A -85,B 0,C 180,E1 -1620,E2 -1620} C_VEL
LIN {X 0,Y 587.365,Z 271.946,A -85,B 0,C 180,E1 -1622.743,E2 -1622.743} C_VEL
LIN {X 0,Y 587.348,Z 271.946,A -85,B 0,C 180,E1 -1625.493,E2 -1625.493} C_VEL
LIN {X 0,Y 587.356,Z 271.945,A -85,B 0,C 180,E1 -1628.255,E2 -1628.255} C_VEL
LIN {X 0,Y 587.339,Z 271.948,A -85,B 0,C 180,E1 -1631.134,E2 -1631.134} C_VEL
LIN {X 0,Y 587.345,Z 271.951,A -85,B 0,C 180,E1 -1633.846,E2 -1633.846} C_VEL
LIN {X 0,Y 587.35,Z 271.952,A -85,B 0,C 180,E1 -1636.818,E2 -1636.818} C_VEL
LIN {X 0,Y 587.318,Z 271.951,A -85,B 0,C 180,E1 -1638.296,E2 -1638.296} C_VEL
LIN {X 0,Y 586.662,Z 272.033,A -85,B 0,C 180,E1 -1638.868,E2 -1638.868} C_VEL
LIN {X 0,Y 583.832,Z 272.39,A -85,B 0,C 180,E1 -1639.797,E2 -1639.797} C_VEL
LIN {X 0,Y 581.423,Z 272.693,A -85,B 0,C 180,E1 -1640.543,E2 -1640.543} C_VEL
LIN {X 0,Y 580.37,Z 272.822,A -85,B 0,C 180,E1 -1641.12,E2 -1641.12} C_VEL
LIN {X 0,Y 580.274,Z 272.831,A -85,B 0,C 180,E1 -1641.315,E2 -1641.315} C_VEL
LIN {X 0,Y 580.273,Z 272.827,A -85,B 0,C 180,E1 -1643.558,E2 -1643.558} C_VEL
LIN {X 0,Y 580.288,Z 272.829,A -85,B 0,C 180,E1 -1645.849,E2 -1645.849} C_VEL
LIN {X 0,Y 580.283,Z 272.826,A -85,B 0,C 180,E1 -1648.187,E2 -1648.187} C_VEL
LIN {X 0,Y 580.286,Z 272.83,A -85,B 0,C 180,E1 -1650.697,E2 -1650.697} C_VEL
LIN {X 0,Y 580.297,Z 272.826,A -85,B 0,C 180,E1 -1653.317,E2 -1653.317} C_VEL
LIN {X 0,Y 580.224,Z 272.833,A -85,B 0,C 180,E1 -1655.755,E2 -1655.755} C_VEL
LIN {X 0,Y 580.285,Z 272.83,A -85,B 0,C 180,E1 -1658.147,E2 -1658.147} C_VEL
LIN {X 0,Y 580.293,Z 272.826,A -85,B 0,C 180,E1 -1660.844,E2 -1660.844} C_VEL
LIN {X 0,Y 580.273,Z 272.827,A -85,B 0,C 180,E1 -1663.659,E2 -1663.659} C_VEL
LIN {X 0,Y 580.281,Z 272.827,A -85,B 0,C 180,E1 -1666.609,E2 -1666.609} C_VEL
LIN {X 0,Y 580.257,Z 272.832,A -85,B 0,C 180,E1 -1668.23,E2 -1668.23} C_VEL
LIN {X 0,Y 580.347,Z 274.97,A -85,B 0,C 180,E1 -1669.723,E2 -1669.723} C_VEL
LIN {X 0,Y 580.303,Z 280.006,A -85,B 0,C 180,E1 -1672.733,E2 -1672.733} C_VEL
LIN {X 0,Y 580.304,Z 284.7,A -85,B 0,C 180,E1 -1675.441,E2 -1675.441} C_VEL
LIN {X 0,Y 580.25,Z 289.247,A -85,B 0,C 180,E1 -1677.978,E2 -1677.978} C_VEL
LIN {X 0,Y 580.222,Z 294.802,A -85,B 0,C 180,E1 -1681.021,E2 -1681.021} C_VEL
LIN {X 0,Y 580.147,Z 299.873,A -85,B 0,C 180,E1 -1683.695,E2 -1683.695} C_VEL
LIN {X 0,Y 580.106,Z 305.213,A -85,B 0,C 180,E1 -1686.435,E2 -1686.435} C_VEL
LIN {X 0,Y 580.074,Z 311.178,A -85,B 0,C 180,E1 -1689.43,E2 -1689.43} C_VEL
LIN {X 0,Y 580.084,Z 315.652,A -85,B 0,C 180,E1 -1691.64,E2 -1691.64} C_VEL
LIN {X 0,Y 580.109,Z 317.837,A -85,B 0,C 180,E1 -1692.668,E2 -1692.668} C_VEL
LIN {X 0,Y 581.534,Z 324.833,A -85,B 0,C 180,E1 -1692.816,E2 -1692.816} C_VEL
LIN {X 0,Y 581.435,Z 339.963,A -85,B 0,C 180,E1 -1693.137,E2 -1693.137} C_VEL
LIN {X 0,Y 581.251,Z 354.526,A -85,B 0,C 180,E1 -1693.583,E2 -1693.583} C_VEL
LIN {X 0,Y 581.104,Z 367.822,A -85,B 0,C 180,E1 -1694.12,E2 -1694.12} C_VEL
LIN {X 0,Y 580.945,Z 381.897,A -85,B 0,C 180,E1 -1694.835,E2 -1694.835} C_VEL
LIN {X 0,Y 580.79,Z 395.741,A -85,B 0,C 180,E1 -1695.706,E2 -1695.706} C_VEL
LIN {X 0,Y 580.61,Z 408.761,A -85,B 0,C 180,E1 -1696.704,E2 -1696.704} C_VEL
LIN {X 0,Y 580.479,Z 420.303,A -85,B 0,C 180,E1 -1697.768,E2 -1697.768} C_VEL
LIN {X 0,Y 580.323,Z 431.001,A -85,B 0,C 180,E1 -1698.945,E2 -1698.945} C_VEL
LIN {X 0,Y 580.27,Z 439.543,A -85,B 0,C 180,E1 -1700.062,E2 -1700.062} C_VEL
LIN {X 0,Y 580.215,Z 447.473,A -85,B 0,C 180,E1 -1701.292,E2 -1701.292} C_VEL
LIN {X 0,Y 580.131,Z 454.882,A -85,B 0,C 180,E1 -1702.692,E2 -1702.692} C_VEL
LIN {X 0,Y 580.132,Z 460.766,A -85,B 0,C 180,E1 -1704.09,E2 -1704.09} C_VEL
LIN {X 0,Y 580.039,Z 464.249,A -85,B 0,C 180,E1 -1705.135,E2 -1705.135} C_VEL
LIN {X 0,Y 580.104,Z 467.794,A -85,B 0,C 180,E1 -1706.527,E2 -1706.527} C_VEL
LIN {X 0,Y 580.039,Z 470.14,A -85,B 0,C 180,E1 -1707.917,E2 -1707.917} C_VEL
LIN {X 0,Y 580.036,Z 471.337,A -85,B 0,C 180,E1 -1709.306,E2 -1709.306} C_VEL
LIN {X 0,Y 580.037,Z 471.36,A -85,B 0,C 180,E1 -1710.694,E2 -1710.694} C_VEL
LIN {X 0,Y 580.039,Z 470.244,A -85,B 0,C 180,E1 -1712.083,E2 -1712.083} C_VEL
LIN {X 0,Y 580.106,Z 467.981,A -85,B 0,C 180,E1 -1713.473,E2 -1713.473} C_VEL
LIN {X 0,Y 580.039,Z 464.521,A -85,B 0,C 180,E1 -1714.866,E2 -1714.866} C_VEL
LIN {X 0,Y 580.092,Z 459.789,A -85,B 0,C 180,E1 -1716.26,E2 -1716.26} C_VEL
LIN {X 0,Y 580.166,Z 453.656,A -85,B 0,C 180,E1 -1717.658,E2 -1717.658} C_VEL
LIN {X 0,Y 580.206,Z 445.937,A -85,B 0,C 180,E1 -1719.06,E2 -1719.06} C_VEL
LIN {X 0,Y 580.291,Z 437.696,A -85,B 0,C 180,E1 -1720.291,E2 -1720.291} C_VEL
LIN {X 0,Y 580.379,Z 427.791,A -85,B 0,C 180,E1 -1721.525,E2 -1721.525} C_VEL
LIN {X 0,Y 580.512,Z 417.64,A -85,B 0,C 180,E1 -1722.587,E2 -1722.587} C_VEL
LIN {X 0,Y 580.68,Z 405.565,A -85,B 0,C 180,E1 -1723.651,E2 -1723.651} C_VEL
LIN {X 0,Y 580.85,Z 392.274,A -85,B 0,C 180,E1 -1724.622,E2 -1724.622} C_VEL
LIN {X 0,Y 580.981,Z 378.726,A -85,B 0,C 180,E1 -1725.434,E2 -1725.434} C_VEL
LIN {X 0,Y 581.17,Z 364.833,A -85,B 0,C 180,E1 -1726.104,E2 -1726.104} C_VEL
LIN {X 0,Y 581.353,Z 350.604,A -85,B 0,C 180,E1 -1726.64,E2 -1726.64} C_VEL
LIN {X 0,Y 581.447,Z 335.748,A -85,B 0,C 180,E1 -1727.057,E2 -1727.057} C_VEL
LIN {X 0,Y 581.38,Z 323.56,A -85,B 0,C 180,E1 -1727.298,E2 -1727.298} C_VEL
LIN {X 0,Y 580.092,Z 317.713,A -85,B 0,C 180,E1 -1727.442,E2 -1727.442} C_VEL
LIN {X 0,Y 580.077,Z 312.85,A -85,B 0,C 180,E1 -1729.83,E2 -1729.83} C_VEL
LIN {X 0,Y 580.119,Z 306.882,A -85,B 0,C 180,E1 -1732.81,E2 -1732.81} C_VEL
LIN {X 0,Y 580.145,Z 300.913,A -85,B 0,C 180,E1 -1735.856,E2 -1735.856} C_VEL
LIN {X 0,Y 580.175,Z 296.45,A -85,B 0,C 180,E1 -1738.192,E2 -1738.192} C_VEL
LIN {X 0,Y 580.231,Z 290.553,A -85,B 0,C 180,E1 -1741.388,E2 -1741.388} C_VEL
LIN {X 0,Y 580.291,Z 286.112,A -85,B 0,C 180,E1 -1743.856,E2 -1743.856} C_VEL
LIN {X 0,Y 580.319,Z 281.659,A -85,B 0,C 180,E1 -1746.4,E2 -1746.4} C_VEL
LIN {X 0,Y 580.317,Z 276.924,A -85,B 0,C 180,E1 -1749.188,E2 -1749.188} C_VEL
LIN {X 0,Y 580.292,Z 273.41,A -85,B 0,C 180,E1 -1751.332,E2 -1751.332} C_VEL
LIN {X 0,Y 580.257,Z 272.834,A -85,B 0,C 180,E1 -1751.77,E2 -1751.77} C_VEL
LIN {X 0,Y 580.266,Z 272.83,A -85,B 0,C 180,E1 -1754.626,E2 -1754.626} C_VEL
LIN {X 0,Y 580.284,Z 272.828,A -85,B 0,C 180,E1 -1757.628,E2 -1757.628} C_VEL
LIN {X 0,Y 580.292,Z 272.828,A -85,B 0,C 180,E1 -1760.067,E2 -1760.067} C_VEL
LIN {X 0,Y 580.297,Z 272.827,A -85,B 0,C 180,E1 -1763.065,E2 -1763.065} C_VEL
LIN {X 0,Y 580.308,Z 272.826,A -85,B 0,C 180,E1 -1766.145,E2 -1766.145} C_VEL
LIN {X 0,Y 580.284,Z 272.826,A -85,B 0,C 180,E1 -1768.615,E2 -1768.615} C_VEL
LIN {X 0,Y 580.284,Z 272.832,A -85,B 0,C 180,E1 -1771.023,E2 -1771.023} C_VEL
LIN {X 0,Y 580.276,Z 272.832,A -85,B 0,C 180,E1 -1774.15,E2 -1774.15} C_VEL
LIN {X 0,Y 580.277,Z 272.827,A -85,B 0,C 180,E1 -1776.442,E2 -1776.442} C_VEL
LIN {X 0,Y 580.261,Z 272.829,A -85,B 0,C 180,E1 -1779.437,E2 -1779.437} C_VEL
LIN {X 0,Y 580.274,Z 272.832,A -85,B 0,C 180,E1 -1781.645,E2 -1781.645} C_VEL
LIN {X 0,Y 580.275,Z 272.827,A -85,B 0,C 180,E1 -1783.825,E2 -1783.825} C_VEL
LIN {X 0,Y 580.252,Z 272.83,A -85,B 0,C 180,E1 -1786.695,E2 -1786.695} C_VEL
LIN {X 0,Y 580.3,Z 272.824,A -85,B 0,C 180,E1 -1788.827,E2 -1788.827} C_VEL
LIN {X 0,Y 580.323,Z 272.821,A -85,B 0,C 180,E1 -1791.644,E2 -1791.644} C_VEL
LIN {X 0,Y 580.316,Z 272.823,A -85,B 0,C 180,E1 -1794.44,E2 -1794.44} C_VEL
LIN {X 0,Y 580.334,Z 272.822,A -85,B 0,C 180,E1 -1797.223,E2 -1797.223} C_VEL
LIN {X 0,Y 580.348,Z 272.823,A -85,B 0,C 180,E1 -1800,E2 -1800} C_VEL
LIN {X 0,Y 580.332,Z 272.822,A -85,B 0,C 180,E1 -1802.776,E2 -1802.776} C_VEL
LIN {X 0,Y 580.318,Z 272.822,A -85,B 0,C 180,E1 -1805.56,E2 -1805.56} C_VEL
LIN {X 0,Y 580.321,Z 272.821,A -85,B 0,C 180,E1 -1808.356,E2 -1808.356} C_VEL
LIN {X 0,Y 580.295,Z 272.826,A -85,B 0,C 180,E1 -1811.191,E2 -1811.191} C_VEL
LIN {X 0,Y 580.308,Z 272.826,A -85,B 0,C 180,E1 -1814.017,E2 -1814.017} C_VEL
LIN {X 0,Y 580.308,Z 272.828,A -85,B 0,C 180,E1 -1816.914,E2 -1816.914} C_VEL
LIN {X 0,Y 580.278,Z 272.831,A -85,B 0,C 180,E1 -1819.823,E2 -1819.823} C_VEL
LIN {X 0,Y 580.26,Z 272.829,A -85,B 0,C 180,E1 -1822.053,E2 -1822.053} C_VEL
LIN {X 0,Y 580.304,Z 272.823,A -85,B 0,C 180,E1 -1825.08,E2 -1825.08} C_VEL
LIN {X 0,Y 580.284,Z 272.826,A -85,B 0,C 180,E1 -1828.186,E2 -1828.186} C_VEL
LIN {X 0,Y 580.282,Z 272.832,A -85,B 0,C 180,E1 -1830.695,E2 -1830.695} C_VEL
LIN {X 0,Y 580.3,Z 272.826,A -85,B 0,C 180,E1 -1833.317,E2 -1833.317} C_VEL
LIN {X 0,Y 580.226,Z 272.835,A -85,B 0,C 180,E1 -1835.754,E2 -1835.754} C_VEL
LIN {X 0,Y 580.287,Z 272.831,A -85,B 0,C 180,E1 -1838.146,E2 -1838.146} C_VEL
LIN {X 0,Y 580.295,Z 272.826,A -85,B 0,C 180,E1 -1840.844,E2 -1840.844} C_VEL
LIN {X 0,Y 580.275,Z 272.828,A -85,B 0,C 180,E1 -1843.658,E2 -1843.658} C_VEL
LIN {X 0,Y 580.275,Z 272.829,A -85,B 0,C 180,E1 -1846.61,E2 -1846.61} C_VEL
LIN {X 0,Y 580.301,Z 272.863,A -85,B 0,C 180,E1 -1848.083,E2 -1848.083} C_VEL
LIN {X 0,Y 580.439,Z 276.688,A -85,B 0,C 180,E1 -1850.08,E2 -1850.08} C_VEL
LIN {X 0,Y 580.374,Z 282.008,A -85,B 0,C 180,E1 -1852.738,E2 -1852.738} C_VEL
LIN {X 0,Y 580.342,Z 287.318,A -85,B 0,C 180,E1 -1855.308,E2 -1855.308} C_VEL
LIN {X 0,Y 580.313,Z 293.047,A -85,B 0,C 180,E1 -1857.968,E2 -1857.968} C_VEL
LIN {X 0,Y 580.263,Z 299.105,A -85,B 0,C 180,E1 -1860.697,E2 -1860.697} C_VEL
LIN {X 0,Y 580.227,Z 305.881,A -85,B 0,C 180,E1 -1863.679,E2 -1863.679} C_VEL
LIN {X 0,Y 580.145,Z 312.275,A -85,B 0,C 180,E1 -1866.436,E2 -1866.436} C_VEL
LIN {X 0,Y 580.151,Z 318.03,A -85,B 0,C 180,E1 -1868.873,E2 -1868.873} C_VEL
LIN {X 0,Y 580.116,Z 324.685,A -85,B 0,C 180,E1 -1871.64,E2 -1871.64} C_VEL
LIN {X 0,Y 580.115,Z 327.076,A -85,B 0,C 180,E1 -1872.614,E2 -1872.614} C_VEL
LIN {X 0,Y 581.519,Z 333.294,A -85,B 0,C 180,E1 -1872.747,E2 -1872.747} C_VEL
LIN {X 0,Y 581.411,Z 348.746,A -85,B 0,C 180,E1 -1873.061,E2 -1873.061} C_VEL
LIN {X 0,Y 581.31,Z 363.207,A -85,B 0,C 180,E1 -1873.494,E2 -1873.494} C_VEL
LIN {X 0,Y 581.119,Z 376.823,A -85,B 0,C 180,E1 -1874.03,E2 -1874.03} C_VEL
LIN {X 0,Y 580.959,Z 391.103,A -85,B 0,C 180,E1 -1874.745,E2 -1874.745} C_VEL
LIN {X 0,Y 580.8,Z 404.568,A -85,B 0,C 180,E1 -1875.58,E2 -1875.58} C_VEL
LIN {X 0,Y 580.629,Z 417.164,A -85,B 0,C 180,E1 -1876.526,E2 -1876.526} C_VEL
LIN {X 0,Y 580.516,Z 428.971,A -85,B 0,C 180,E1 -1877.591,E2 -1877.591} C_VEL
LIN {X 0,Y 580.336,Z 440.089,A -85,B 0,C 180,E1 -1878.792,E2 -1878.792} C_VEL
LIN {X 0,Y 580.268,Z 449.856,A -85,B 0,C 180,E1 -1880.061,E2 -1880.061} C_VEL
LIN {X 0,Y 580.215,Z 457.731,A -85,B 0,C 180,E1 -1881.291,E2 -1881.291} C_VEL
LIN {X 0,Y 580.13,Z 465.088,A -85,B 0,C 180,E1 -1882.692,E2 -1882.692} C_VEL
LIN {X 0,Y 580.132,Z 470.923,A -85,B 0,C 180,E1 -1884.089,E2 -1884.089} C_VEL
LIN {X 0,Y 580.041,Z 474.384,A -85,B 0,C 180,E1 -1885.134,E2 -1885.134} C_VEL
LIN {X 0,Y 580.105,Z 477.888,A -85,B 0,C 180,E1 -1886.527,E2 -1886.527} C_VEL
LIN {X 0,Y 580.039,Z 480.193,A -85,B 0,C 180,E1 -1887.917,E2 -1887.917} C_VEL
LIN {X 0,Y 580.036,Z 481.349,A -85,B 0,C 180,E1 -1889.306,E2 -1889.306} C_VEL
LIN {X 0,Y 580.036,Z 481.349,A -85,B 0,C 180,E1 -1890.694,E2 -1890.694} C_VEL
LIN {X 0,Y 580.039,Z 480.192,A -85,B 0,C 180,E1 -1892.083,E2 -1892.083} C_VEL
LIN {X 0,Y 580.105,Z 477.887,A -85,B 0,C 180,E1 -1893.473,E2 -1893.473} C_VEL
LIN {X 0,Y 580.041,Z 474.386,A -85,B 0,C 180,E1 -1894.865,E2 -1894.865} C_VEL
LIN {X 0,Y 580.093,Z 469.61,A -85,B 0,C 180,E1 -1896.259,E2 -1896.259} C_VEL
LIN {X 0,Y 580.165,Z 463.426,A -85,B 0,C 180,E1 -1897.657,E2 -1897.657} C_VEL
LIN {X 0,Y 580.207,Z 455.653,A -85,B 0,C 180,E1 -1899.06,E2 -1899.06} C_VEL
LIN {X 0,Y 580.308,Z 447.373,A -85,B 0,C 180,E1 -1900.29,E2 -1900.29} C_VEL
LIN {X 0,Y 580.382,Z 437.399,A -85,B 0,C 180,E1 -1901.525,E2 -1901.525} C_VEL
LIN {X 0,Y 580.541,Z 427.195,A -85,B 0,C 180,E1 -1902.586,E2 -1902.586} C_VEL
LIN {X 0,Y 580.677,Z 415.024,A -85,B 0,C 180,E1 -1903.651,E2 -1903.651} C_VEL
LIN {X 0,Y 580.845,Z 402.813,A -85,B 0,C 180,E1 -1904.541,E2 -1904.541} C_VEL
LIN {X 0,Y 580.963,Z 389.528,A -85,B 0,C 180,E1 -1905.344,E2 -1905.344} C_VEL
LIN {X 0,Y 581.169,Z 374.847,A -85,B 0,C 180,E1 -1906.058,E2 -1906.058} C_VEL
LIN {X 0,Y 581.306,Z 360.632,A -85,B 0,C 180,E1 -1906.596,E2 -1906.596} C_VEL
LIN {X 0,Y 581.461,Z 345.94,A -85,B 0,C 180,E1 -1907.007,E2 -1907.007} C_VEL
LIN {X 0,Y 581.405,Z 332.784,A -85,B 0,C 180,E1 -1907.264,E2 -1907.264} C_VEL
LIN {X 0,Y 580.137,Z 326.99,A -85,B 0,C 180,E1 -1907.411,E2 -1907.411} C_VEL
LIN {X 0,Y 580.12,Z 321.14,A -85,B 0,C 180,E1 -1909.828,E2 -1909.828} C_VEL
LIN {X 0,Y 580.16,Z 315.822,A -85,B 0,C 180,E1 -1912.056,E2 -1912.056} C_VEL
LIN {X 0,Y 580.159,Z 308.731,A -85,B 0,C 180,E1 -1915.086,E2 -1915.086} C_VEL
LIN {X 0,Y 580.225,Z 303.413,A -85,B 0,C 180,E1 -1917.404,E2 -1917.404} C_VEL
LIN {X 0,Y 580.259,Z 298.047,A -85,B 0,C 180,E1 -1919.773,E2 -1919.773} C_VEL
LIN {X 0,Y 580.311,Z 292.684,A -85,B 0,C 180,E1 -1922.199,E2 -1922.199} C_VEL
LIN {X 0,Y 580.34,Z 287.32,A -85,B 0,C 180,E1 -1924.692,E2 -1924.692} C_VEL
LIN {X 0,Y 580.389,Z 282.009,A -85,B 0,C 180,E1 -1927.261,E2 -1927.261} C_VEL
LIN {X 0,Y 580.463,Z 275.96,A -85,B 0,C 180,E1 -1930.291,E2 -1930.291} C_VEL
LIN {X 0,Y 580.291,Z 272.83,A -85,B 0,C 180,E1 -1931.992,E2 -1931.992} C_VEL
LIN {X 0,Y 580.263,Z 272.83,A -85,B 0,C 180,E1 -1934.625,E2 -1934.625} C_VEL
LIN {X 0,Y 580.279,Z 272.828,A -85,B 0,C 180,E1 -1937.628,E2 -1937.628} C_VEL
LIN {X 0,Y 580.29,Z 272.83,A -85,B 0,C 180,E1 -1940.067,E2 -1940.067} C_VEL
LIN {X 0,Y 580.292,Z 272.828,A -85,B 0,C 180,E1 -1943.065,E2 -1943.065} C_VEL
LIN {X 0,Y 580.305,Z 272.827,A -85,B 0,C 180,E1 -1946.145,E2 -1946.145} C_VEL
LIN {X 0,Y 580.282,Z 272.827,A -85,B 0,C 180,E1 -1948.615,E2 -1948.615} C_VEL
LIN {X 0,Y 580.28,Z 272.832,A -85,B 0,C 180,E1 -1951.023,E2 -1951.023} C_VEL
LIN {X 0,Y 580.284,Z 272.828,A -85,B 0,C 180,E1 -1953.665,E2 -1953.665} C_VEL
LIN {X 0,Y 580.293,Z 272.828,A -85,B 0,C 180,E1 -1955.684,E2 -1955.684} C_VEL
LIN {X 0,Y 580.259,Z 272.829,A -85,B 0,C 180,E1 -1957.947,E2 -1957.947} C_VEL
LIN {X 0,Y 580.31,Z 272.822,A -85,B 0,C 180,E1 -1960.914,E2 -1960.914} C_VEL
LIN {X 0,Y 580.27,Z 272.828,A -85,B 0,C 180,E1 -1963.825,E2 -1963.825} C_VEL
LIN {X 0,Y 580.258,Z 272.83,A -85,B 0,C 180,E1 -1966.696,E2 -1966.696} C_VEL
LIN {X 0,Y 580.301,Z 272.827,A -85,B 0,C 180,E1 -1969.533,E2 -1969.533} C_VEL
LIN {X 0,Y 580.308,Z 272.829,A -85,B 0,C 180,E1 -1972.344,E2 -1972.344} C_VEL
LIN {X 0,Y 580.332,Z 272.822,A -85,B 0,C 180,E1 -1975.137,E2 -1975.137} C_VEL
LIN {X 0,Y 580.341,Z 272.819,A -85,B 0,C 180,E1 -1977.918,E2 -1977.918} C_VEL
LIN {X 0,Y 580.337,Z 272.819,A -85,B 0,C 180,E1 -1980.694,E2 -1980.694} C_VEL
LIN {X 0,Y 580.286,Z 272.827,A -85,B 0,C 180,E1 -1983.472,E2 -1983.472} C_VEL
LIN {X 0,Y 580.316,Z 272.822,A -85,B 0,C 180,E1 -1985.56,E2 -1985.56} C_VEL
LIN {X 0,Y 580.319,Z 272.821,A -85,B 0,C 180,E1 -1988.356,E2 -1988.356} C_VEL
LIN {X 0,Y 580.291,Z 272.825,A -85,B 0,C 180,E1 -1991.191,E2 -1991.191} C_VEL
LIN {X 0,Y 580.303,Z 272.826,A -85,B 0,C 180,E1 -1994.018,E2 -1994.018} C_VEL
LIN {X 0,Y 580.303,Z 272.828,A -85,B 0,C 180,E1 -1996.914,E2 -1996.914} C_VEL
LIN {X 0,Y 580.291,Z 272.83,A -85,B 0,C 180,E1 -1999.823,E2 -1999.823} C_VEL
LIN {X 0,Y 580.274,Z 272.831,A -85,B 0,C 180,E1 -2001.315,E2 -2001.315} C_VEL
LIN {X 0,Y 579.575,Z 272.916,A -85,B 0,C 180,E1 -2001.894,E2 -2001.894} C_VEL
LIN {X 0,Y 576.7,Z 273.277,A -85,B 0,C 180,E1 -2002.834,E2 -2002.834} C_VEL
LIN {X 0,Y 574.307,Z 273.572,A -85,B 0,C 180,E1 -2003.59,E2 -2003.59} C_VEL
LIN {X 0,Y 573.309,Z 273.697,A -85,B 0,C 180,E1 -2004.174,E2 -2004.174} C_VEL
LIN {X 0,Y 573.242,Z 273.704,A -85,B 0,C 180,E1 -2004.372,E2 -2004.372} C_VEL
LIN {X 0,Y 573.24,Z 273.703,A -85,B 0,C 180,E1 -2006.977,E2 -2006.977} C_VEL
LIN {X 0,Y 573.237,Z 273.704,A -85,B 0,C 180,E1 -2009.488,E2 -2009.488} C_VEL
LIN {X 0,Y 573.249,Z 273.706,A -85,B 0,C 180,E1 -2012.23,E2 -2012.23} C_VEL
LIN {X 0,Y 573.219,Z 273.707,A -85,B 0,C 180,E1 -2014.771,E2 -2014.771} C_VEL
LIN {X 0,Y 573.232,Z 273.705,A -85,B 0,C 180,E1 -2017.808,E2 -2017.808} C_VEL
LIN {X 0,Y 573.264,Z 273.701,A -85,B 0,C 180,E1 -2020.529,E2 -2020.529} C_VEL
LIN {X 0,Y 573.238,Z 273.704,A -85,B 0,C 180,E1 -2023.67,E2 -2023.67} C_VEL
LIN {X 0,Y 573.242,Z 273.704,A -85,B 0,C 180,E1 -2026.642,E2 -2026.642} C_VEL
LIN {X 0,Y 573.219,Z 273.867,A -85,B 0,C 180,E1 -2028.409,E2 -2028.409} C_VEL
LIN {X 0,Y 573.293,Z 277.328,A -85,B 0,C 180,E1 -2030.563,E2 -2030.563} C_VEL
LIN {X 0,Y 573.282,Z 281.521,A -85,B 0,C 180,E1 -2033.081,E2 -2033.081} C_VEL
LIN {X 0,Y 573.266,Z 285.98,A -85,B 0,C 180,E1 -2035.672,E2 -2035.672} C_VEL
LIN {X 0,Y 573.181,Z 290.433,A -85,B 0,C 180,E1 -2038.182,E2 -2038.182} C_VEL
LIN {X 0,Y 573.15,Z 296.323,A -85,B 0,C 180,E1 -2041.432,E2 -2041.432} C_VEL
LIN {X 0,Y 573.082,Z 302.233,A -85,B 0,C 180,E1 -2044.582,E2 -2044.582} C_VEL
LIN {X 0,Y 573.012,Z 308.197,A -85,B 0,C 180,E1 -2047.654,E2 -2047.654} C_VEL
LIN {X 0,Y 573.017,Z 314.162,A -85,B 0,C 180,E1 -2050.662,E2 -2050.662} C_VEL
LIN {X 0,Y 573.025,Z 317.826,A -85,B 0,C 180,E1 -2052.446,E2 -2052.446} C_VEL
LIN {X 0,Y 574.751,Z 326.014,A -85,B 0,C 180,E1 -2052.624,E2 -2052.624} C_VEL
LIN {X 0,Y 574.629,Z 341.774,A -85,B 0,C 180,E1 -2052.977,E2 -2052.977} C_VEL
LIN {X 0,Y 574.395,Z 357.165,A -85,B 0,C 180,E1 -2053.477,E2 -2053.477} C_VEL
LIN {X 0,Y 574.212,Z 371.737,A -85,B 0,C 180,E1 -2054.107,E2 -2054.107} C_VEL
LIN {X 0,Y 574.031,Z 385.041,A -85,B 0,C 180,E1 -2054.83,E2 -2054.83} C_VEL
LIN {X 0,Y 573.858,Z 398.56,A -85,B 0,C 180,E1 -2055.729,E2 -2055.729} C_VEL
LIN {X 0,Y 573.629,Z 410.886,A -85,B 0,C 180,E1 -2056.72,E2 -2056.72} C_VEL
LIN {X 0,Y 573.458,Z 422.084,A -85,B 0,C 180,E1 -2057.796,E2 -2057.796} C_VEL
LIN {X 0,Y 573.294,Z 431.585,A -85,B 0,C 180,E1 -2058.877,E2 -2058.877} C_VEL
LIN {X 0,Y 573.202,Z 440.78,A -85,B 0,C 180,E1 -2060.116,E2 -2060.116} C_VEL
LIN {X 0,Y 573.134,Z 448.488,A -85,B 0,C 180,E1 -2061.361,E2 -2061.361} C_VEL
LIN {X 0,Y 573.075,Z 454.884,A -85,B 0,C 180,E1 -2062.602,E2 -2062.602} C_VEL
LIN {X 0,Y 573.042,Z 460.768,A -85,B 0,C 180,E1 -2064.017,E2 -2064.017} C_VEL
LIN {X 0,Y 572.949,Z 464.251,A -85,B 0,C 180,E1 -2065.075,E2 -2065.075} C_VEL
LIN {X 0,Y 573.004,Z 467.796,A -85,B 0,C 180,E1 -2066.484,E2 -2066.484} C_VEL
LIN {X 0,Y 572.938,Z 470.14,A -85,B 0,C 180,E1 -2067.891,E2 -2067.891} C_VEL
LIN {X 0,Y 572.936,Z 471.337,A -85,B 0,C 180,E1 -2069.297,E2 -2069.297} C_VEL
LIN {X 0,Y 572.937,Z 471.359,A -85,B 0,C 180,E1 -2070.703,E2 -2070.703} C_VEL
LIN {X 0,Y 572.939,Z 470.243,A -85,B 0,C 180,E1 -2072.109,E2 -2072.109} C_VEL
LIN {X 0,Y 573.006,Z 467.98,A -85,B 0,C 180,E1 -2073.516,E2 -2073.516} C_VEL
LIN {X 0,Y 572.949,Z 464.52,A -85,B 0,C 180,E1 -2074.926,E2 -2074.926} C_VEL
LIN {X 0,Y 573.007,Z 459.787,A -85,B 0,C 180,E1 -2076.338,E2 -2076.338} C_VEL
LIN {X 0,Y 573.094,Z 453.653,A -85,B 0,C 180,E1 -2077.753,E2 -2077.753} C_VEL
LIN {X 0,Y 573.134,Z 445.933,A -85,B 0,C 180,E1 -2079.173,E2 -2079.173} C_VEL
LIN {X 0,Y 573.265,Z 437.692,A -85,B 0,C 180,E1 -2080.418,E2 -2080.418} C_VEL
LIN {X 0,Y 573.354,Z 427.783,A -85,B 0,C 180,E1 -2081.669,E2 -2081.669} C_VEL
LIN {X 0,Y 573.534,Z 417.634,A -85,B 0,C 180,E1 -2082.743,E2 -2082.743} C_VEL
LIN {X 0,Y 573.722,Z 405.556,A -85,B 0,C 180,E1 -2083.82,E2 -2083.82} C_VEL
LIN {X 0,Y 573.929,Z 392.67,A -85,B 0,C 180,E1 -2084.775,E2 -2084.775} C_VEL
LIN {X 0,Y 574.111,Z 378.716,A -85,B 0,C 180,E1 -2085.623,E2 -2085.623} C_VEL
LIN {X 0,Y 574.322,Z 364.818,A -85,B 0,C 180,E1 -2086.301,E2 -2086.301} C_VEL
LIN {X 0,Y 574.543,Z 350.585,A -85,B 0,C 180,E1 -2086.843,E2 -2086.843} C_VEL
LIN {X 0,Y 574.66,Z 335.723,A -85,B 0,C 180,E1 -2087.265,E2 -2087.265} C_VEL
LIN {X 0,Y 574.599,Z 324.698,A -85,B 0,C 180,E1 -2087.491,E2 -2087.491} C_VEL
LIN {X 0,Y 573.007,Z 317.735,A -85,B 0,C 180,E1 -2087.653,E2 -2087.653} C_VEL
LIN {X 0,Y 572.991,Z 312.849,A -85,B 0,C 180,E1 -2090.086,E2 -2090.086} C_VEL
LIN {X 0,Y 573.073,Z 306.881,A -85,B 0,C 180,E1 -2093.106,E2 -2093.106} C_VEL
LIN {X 0,Y 573.08,Z 302.404,A -85,B 0,C 180,E1 -2095.418,E2 -2095.418} C_VEL
LIN {X 0,Y 573.134,Z 297.527,A -85,B 0,C 180,E1 -2098.006,E2 -2098.006} C_VEL
LIN {X 0,Y 573.156,Z 292.062,A -85,B 0,C 180,E1 -2100.997,E2 -2100.997} C_VEL
LIN {X 0,Y 573.241,Z 287.551,A -85,B 0,C 180,E1 -2103.52,E2 -2103.52} C_VEL
LIN {X 0,Y 573.299,Z 283.165,A -85,B 0,C 180,E1 -2106.045,E2 -2106.045} C_VEL
LIN {X 0,Y 573.268,Z 278.699,A -85,B 0,C 180,E1 -2108.699,E2 -2108.699} C_VEL
LIN {X 0,Y 573.327,Z 275.69,A -85,B 0,C 180,E1 -2110.535,E2 -2110.535} C_VEL
LIN {X 0,Y 573.23,Z 274.006,A -85,B 0,C 180,E1 -2111.593,E2 -2111.593} C_VEL
LIN {X 0,Y 573.238,Z 273.705,A -85,B 0,C 180,E1 -2113.359,E2 -2113.359} C_VEL
LIN {X 0,Y 573.242,Z 273.704,A -85,B 0,C 180,E1 -2116.331,E2 -2116.331} C_VEL
LIN {X 0,Y 573.222,Z 273.709,A -85,B 0,C 180,E1 -2118.542,E2 -2118.542} C_VEL
LIN {X 0,Y 573.249,Z 273.703,A -85,B 0,C 180,E1 -2121.299,E2 -2121.299} C_VEL
LIN {X 0,Y 573.188,Z 273.71,A -85,B 0,C 180,E1 -2124.021,E2 -2124.021} C_VEL
LIN {X 0,Y 573.267,Z 273.705,A -85,B 0,C 180,E1 -2126.518,E2 -2126.518} C_VEL
LIN {X 0,Y 573.235,Z 273.706,A -85,B 0,C 180,E1 -2129.116,E2 -2129.116} C_VEL
LIN {X 0,Y 573.22,Z 273.707,A -85,B 0,C 180,E1 -2131.434,E2 -2131.434} C_VEL
LIN {X 0,Y 573.246,Z 273.703,A -85,B 0,C 180,E1 -2134.589,E2 -2134.589} C_VEL
LIN {X 0,Y 573.23,Z 273.704,A -85,B 0,C 180,E1 -2137.662,E2 -2137.662} C_VEL
LIN {X 0,Y 573.261,Z 273.701,A -85,B 0,C 180,E1 -2140.67,E2 -2140.67} C_VEL
LIN {X 0,Y 573.247,Z 273.703,A -85,B 0,C 180,E1 -2143.622,E2 -2143.622} C_VEL
LIN {X 0,Y 573.211,Z 273.709,A -85,B 0,C 180,E1 -2146.529,E2 -2146.529} C_VEL
LIN {X 0,Y 573.259,Z 273.701,A -85,B 0,C 180,E1 -2148.745,E2 -2148.745} C_VEL
LIN {X 0,Y 573.279,Z 273.698,A -85,B 0,C 180,E1 -2151.54,E2 -2151.54} C_VEL
LIN {X 0,Y 573.283,Z 273.699,A -85,B 0,C 180,E1 -2154.372,E2 -2154.372} C_VEL
LIN {X 0,Y 573.313,Z 273.694,A -85,B 0,C 180,E1 -2157.892,E2 -2157.892} C_VEL
LIN {X 0,Y 573.312,Z 273.694,A -85,B 0,C 180,E1 -2160.702,E2 -2160.702} C_VEL
LIN {X 0,Y 573.3,Z 273.698,A -85,B 0,C 180,E1 -2162.811,E2 -2162.811} C_VEL
LIN {X 0,Y 573.286,Z 273.698,A -85,B 0,C 180,E1 -2165.628,E2 -2165.628} C_VEL
LIN {X 0,Y 573.278,Z 273.699,A -85,B 0,C 180,E1 -2168.46,E2 -2168.46} C_VEL
LIN {X 0,Y 573.267,Z 273.7,A -85,B 0,C 180,E1 -2171.312,E2 -2171.312} C_VEL
LIN {X 0,Y 573.252,Z 273.703,A -85,B 0,C 180,E1 -2174.193,E2 -2174.193} C_VEL
LIN {X 0,Y 573.256,Z 273.704,A -85,B 0,C 180,E1 -2177.112,E2 -2177.112} C_VEL
LIN {X 0,Y 573.233,Z 273.708,A -85,B 0,C 180,E1 -2180.077,E2 -2180.077} C_VEL
LIN {X 0,Y 573.226,Z 273.705,A -85,B 0,C 180,E1 -2182.338,E2 -2182.338} C_VEL
LIN {X 0,Y 573.252,Z 273.702,A -85,B 0,C 180,E1 -2185.41,E2 -2185.41} C_VEL
LIN {X 0,Y 573.223,Z 273.706,A -85,B 0,C 180,E1 -2188.565,E2 -2188.565} C_VEL
LIN {X 0,Y 573.228,Z 273.707,A -85,B 0,C 180,E1 -2190.993,E2 -2190.993} C_VEL
LIN {X 0,Y 573.259,Z 273.706,A -85,B 0,C 180,E1 -2193.524,E2 -2193.524} C_VEL
LIN {X 0,Y 573.249,Z 273.707,A -85,B 0,C 180,E1 -2196.923,E2 -2196.923} C_VEL
LIN {X 0,Y 573.246,Z 273.707,A -85,B 0,C 180,E1 -2199.607,E2 -2199.607} C_VEL
LIN {X 0,Y 573.226,Z 273.709,A -85,B 0,C 180,E1 -2202.64,E2 -2202.64} C_VEL
LIN {X 0,Y 573.234,Z 273.71,A -85,B 0,C 180,E1 -2205.667,E2 -2205.667} C_VEL
LIN {X 0,Y 573.264,Z 273.72,A -85,B 0,C 180,E1 -2207.92,E2 -2207.92} C_VEL
LIN {X 0,Y 573.475,Z 276.666,A -85,B 0,C 180,E1 -2209.495,E2 -2209.495} C_VEL
LIN {X 0,Y 573.394,Z 281.979,A -85,B 0,C 180,E1 -2212.205,E2 -2212.205} C_VEL
LIN {X 0,Y 573.325,Z 287.298,A -85,B 0,C 180,E1 -2214.821,E2 -2214.821} C_VEL
LIN {X 0,Y 573.285,Z 292.646,A -85,B 0,C 180,E1 -2217.357,E2 -2217.357} C_VEL
LIN {X 0,Y 573.207,Z 299.553,A -85,B 0,C 180,E1 -2220.519,E2 -2220.519} C_VEL
LIN {X 0,Y 573.164,Z 305.171,A -85,B 0,C 180,E1 -2223.02,E2 -2223.02} C_VEL
LIN {X 0,Y 573.081,Z 312.275,A -85,B 0,C 180,E1 -2226.128,E2 -2226.128} C_VEL
LIN {X 0,Y 573.104,Z 318.375,A -85,B 0,C 180,E1 -2228.747,E2 -2228.747} C_VEL
LIN {X 0,Y 573.038,Z 324.685,A -85,B 0,C 180,E1 -2231.405,E2 -2231.405} C_VEL
LIN {X 0,Y 573.065,Z 327.218,A -85,B 0,C 180,E1 -2232.395,E2 -2232.395} C_VEL
LIN {X 0,Y 574.748,Z 334.74,A -85,B 0,C 180,E1 -2232.559,E2 -2232.559} C_VEL
LIN {X 0,Y 574.635,Z 349.538,A -85,B 0,C 180,E1 -2232.875,E2 -2232.875} C_VEL
LIN {X 0,Y 574.487,Z 364.501,A -85,B 0,C 180,E1 -2233.338,E2 -2233.338} C_VEL
LIN {X 0,Y 574.245,Z 378.8,A -85,B 0,C 180,E1 -2233.925,E2 -2233.925} C_VEL
LIN {X 0,Y 574.043,Z 392.676,A -85,B 0,C 180,E1 -2234.648,E2 -2234.648} C_VEL
LIN {X 0,Y 573.872,Z 405.971,A -85,B 0,C 180,E1 -2235.501,E2 -2235.501} C_VEL
LIN {X 0,Y 573.656,Z 418.229,A -85,B 0,C 180,E1 -2236.449,E2 -2236.449} C_VEL
LIN {X 0,Y 573.511,Z 428.97,A -85,B 0,C 180,E1 -2237.437,E2 -2237.437} C_VEL
LIN {X 0,Y 573.349,Z 438.901,A -85,B 0,C 180,E1 -2238.51,E2 -2238.51} C_VEL
LIN {X 0,Y 573.256,Z 448.619,A -85,B 0,C 180,E1 -2239.76,E2 -2239.76} C_VEL
LIN {X 0,Y 573.135,Z 456.721,A -85,B 0,C 180,E1 -2241.005,E2 -2241.005} C_VEL
LIN {X 0,Y 573.093,Z 463.424,A -85,B 0,C 180,E1 -2242.247,E2 -2242.247} C_VEL
LIN {X 0,Y 573.015,Z 469.606,A -85,B 0,C 180,E1 -2243.662,E2 -2243.662} C_VEL
LIN {X 0,Y 572.951,Z 474.384,A -85,B 0,C 180,E1 -2245.074,E2 -2245.074} C_VEL
LIN {X 0,Y 573.005,Z 477.888,A -85,B 0,C 180,E1 -2246.484,E2 -2246.484} C_VEL
LIN {X 0,Y 572.938,Z 480.192,A -85,B 0,C 180,E1 -2247.891,E2 -2247.891} C_VEL
LIN {X 0,Y 572.936,Z 481.349,A -85,B 0,C 180,E1 -2249.297,E2 -2249.297} C_VEL
LIN {X 0,Y 572.936,Z 481.349,A -85,B 0,C 180,E1 -2250.703,E2 -2250.703} C_VEL
LIN {X 0,Y 572.938,Z 480.191,A -85,B 0,C 180,E1 -2252.109,E2 -2252.109} C_VEL
LIN {X 0,Y 573.005,Z 477.887,A -85,B 0,C 180,E1 -2253.516,E2 -2253.516} C_VEL
LIN {X 0,Y 572.951,Z 474.386,A -85,B 0,C 180,E1 -2254.925,E2 -2254.925} C_VEL
LIN {X 0,Y 573.013,Z 469.61,A -85,B 0,C 180,E1 -2256.337,E2 -2256.337} C_VEL
LIN {X 0,Y 573.093,Z 463.425,A -85,B 0,C 180,E1 -2257.752,E2 -2257.752} C_VEL
LIN {X 0,Y 573.135,Z 455.652,A -85,B 0,C 180,E1 -2259.172,E2 -2259.172} C_VEL
LIN {X 0,Y 573.27,Z 447.372,A -85,B 0,C 180,E1 -2260.418,E2 -2260.418} C_VEL
LIN {X 0,Y 573.385,Z 437.396,A -85,B 0,C 180,E1 -2261.668,E2 -2261.668} C_VEL
LIN {X 0,Y 573.567,Z 427.194,A -85,B 0,C 180,E1 -2262.741,E2 -2262.741} C_VEL
LIN {X 0,Y 573.742,Z 415.025,A -85,B 0,C 180,E1 -2263.819,E2 -2263.819} C_VEL
LIN {X 0,Y 573.961,Z 401.91,A -85,B 0,C 180,E1 -2264.781,E2 -2264.781} C_VEL
LIN {X 0,Y 574.122,Z 387.879,A -85,B 0,C 180,E1 -2265.623,E2 -2265.623} C_VEL
LIN {X 0,Y 574.322,Z 373.81,A -85,B 0,C 180,E1 -2266.301,E2 -2266.301} C_VEL
LIN {X 0,Y 574.563,Z 359.32,A -85,B 0,C 180,E1 -2266.842,E2 -2266.842} C_VEL
LIN {X 0,Y 574.686,Z 343.677,A -85,B 0,C 180,E1 -2267.269,E2 -2267.269} C_VEL
LIN {X 0,Y 574.514,Z 333.362,A -85,B 0,C 180,E1 -2267.469,E2 -2267.469} C_VEL
LIN {X 0,Y 573.048,Z 327.017,A -85,B 0,C 180,E1 -2267.622,E2 -2267.622} C_VEL
LIN {X 0,Y 573.039,Z 321.14,A -85,B 0,C 180,E1 -2270.084,E2 -2270.084} C_VEL
LIN {X 0,Y 573.08,Z 315.822,A -85,B 0,C 180,E1 -2272.344,E2 -2272.344} C_VEL
LIN {X 0,Y 573.106,Z 308.731,A -85,B 0,C 180,E1 -2275.416,E2 -2275.416} C_VEL
LIN {X 0,Y 573.193,Z 302.812,A -85,B 0,C 180,E1 -2278.018,E2 -2278.018} C_VEL
LIN {X 0,Y 573.207,Z 298.011,A -85,B 0,C 180,E1 -2280.178,E2 -2280.178} C_VEL
LIN {X 0,Y 573.283,Z 292.647,A -85,B 0,C 180,E1 -2282.642,E2 -2282.642} C_VEL
LIN {X 0,Y 573.323,Z 287.3,A -85,B 0,C 180,E1 -2285.179,E2 -2285.179} C_VEL
LIN {X 0,Y 573.431,Z 280.901,A -85,B 0,C 180,E1 -2288.336,E2 -2288.336} C_VEL
LIN {X 0,Y 573.464,Z 276.58,A -85,B 0,C 180,E1 -2290.551,E2 -2290.551} C_VEL
